SPLINE
SPL {X  -125.038, Y  +285.873, Z    +0.000, E1   +53.023, E3 +71876.787}
SPL {X  -149.949, Y  +329.886, Z    +0.000, E1   +41.515, E3 +71898.352}
SPL {X  -157.246, Y  +356.141, Z    +0.000, E1   +27.282, E3 +71903.408}
SPL {X  -159.525, Y  +373.376, Z    +0.000, E1   +13.812, E3 +71905.065}
SPL {X  -160.000, Y  +387.264, Z    +0.000, E1    +0.544, E3 +71905.523}
SPL {X  -160.000, Y  +390.384, Z    +0.000, E1    -6.008, E3 +71905.560}
SPL {X  -160.000, Y  +395.752, Z    +0.000, E1   -19.038, E3 +71905.754}
SPL {X  -160.000, Y  +404.289, Z    +0.000, E1   -38.292, E3 +71906.422}
SPL {X  -160.000, Y  +418.681, Z    +0.000, E1   -56.949, E3 +71908.612}
SPL {X  -160.000, Y  +471.977, Z    +0.000, E1   -70.792, E3 +71925.131}
SPL {X  -159.977, Y  +677.138, Z    +0.000, E1   -73.665, E3 +72021.623}
SPL {X  -157.805, Y  +700.810, Z    +0.000, E1   -73.511, E3 +72038.453}
SPL {X  -152.242, Y  +723.618, Z    +0.000, E1   -72.940, E3 +72058.366}
SPL {X  -145.929, Y  +740.010, Z    +0.000, E1   -72.229, E3 +72074.837}
SPL {X  -139.114, Y  +753.439, Z    +0.000, E1   -71.436, E3 +72089.476}
SPL {X  -132.333, Y  +764.333, Z    +0.000, E1   -70.535, E3 +72102.100}
SPL {X  -125.486, Y  +773.664, Z    +0.000, E1   -69.598, E3 +72113.074}
SPL {X  -121.321, Y  +778.713, Z    +0.000, E1   -68.872, E3 +72119.084}
SPL {X   -77.337, Y  +814.468, Z    +0.000, E1   -56.377, E3 +72237.715}
ENDSPLINE

SPLINE
SPL {X  -134.727, Y  +760.706, Z    +0.000, E1   -50.460, E3 +72425.947}
SPL {X  -155.580, Y  +711.748, Z    +0.000, E1   -32.084, E3 +72442.861}
SPL {X  -159.445, Y  +687.715, Z    +0.000, E1   -14.660, E3 +72445.708}
SPL {X  -159.995, Y  +675.725, Z    +0.000, E1    -3.424, E3 +72446.219}
SPL {X  -160.000, Y  +671.714, Z    +0.000, E1    +0.835, E3 +72446.259}
SPL {X  -160.000, Y  +663.084, Z    +0.000, E1   +21.134, E3 +72446.584}
SPL {X  -160.000, Y  +650.910, Z    +0.000, E1   +46.005, E3 +72447.738}
SPL {X  -160.000, Y  +634.843, Z    +0.000, E1   +61.273, E3 +72450.414}
SPL {X  -160.000, Y  +578.679, Z    +0.000, E1   +71.665, E3 +72468.248}
SPL {X  -160.000, Y  +387.528, Z    +0.000, E1   +73.487, E3 +72561.061}
SPL {X  -159.218, Y  +369.903, Z    +0.000, E1   +73.425, E3 +72572.928}
SPL {X  -156.808, Y  +353.900, Z    +0.000, E1   +73.180, E3 +72585.531}
SPL {X  -154.539, Y  +344.254, Z    +0.000, E1   +72.827, E3 +72595.069}
ENDSPLINE

SPLINE
SPL {X  -157.258, Y  +356.206, Z    +0.000, E1   +70.434, E3 +72609.641}
ENDSPLINE

SPLINE
SPL {X  -150.342, Y  +330.952, Z    +0.000, E1   +71.154, E3 +72621.314}
SPL {X  -141.358, Y  +310.748, Z    +0.000, E1   +71.233, E3 +72634.019}
SPL {X  -134.330, Y  +298.778, Z    +0.000, E1   +70.323, E3 +72647.867}
SPL {X  -128.957, Y  +290.989, Z    +0.000, E1   +69.528, E3 +72657.232}
SPL {X  -124.846, Y  +285.632, Z    +0.000, E1   +68.906, E3 +72663.695}
SPL {X  -121.783, Y  +281.927, Z    +0.000, E1   +68.403, E3 +72668.127}
SPL {X   -79.219, Y  +246.688, Z    +0.000, E1   +55.887, E3 +72789.634}
ENDSPLINE

SPLINE
SPL {X  -125.038, Y  +285.873, Z    +0.000, E1   +53.023, E3 +72966.675}
SPL {X  -149.949, Y  +329.886, Z    +0.000, E1   +41.515, E3 +72988.240}
SPL {X  -157.246, Y  +356.141, Z    +0.000, E1   +27.282, E3 +72993.296}
SPL {X  -159.525, Y  +373.376, Z    +0.000, E1   +13.812, E3 +72994.954}
SPL {X  -160.000, Y  +387.264, Z    +0.000, E1    +0.544, E3 +72995.411}
SPL {X  -160.000, Y  +390.384, Z    +0.000, E1    -6.008, E3 +72995.448}
SPL {X  -160.000, Y  +395.752, Z    +0.000, E1   -19.038, E3 +72995.642}
SPL {X  -160.000, Y  +404.289, Z    +0.000, E1   -38.292, E3 +72996.311}
SPL {X  -160.000, Y  +418.681, Z    +0.000, E1   -56.949, E3 +72998.500}
SPL {X  -160.000, Y  +471.977, Z    +0.000, E1   -70.792, E3 +73015.020}
SPL {X  -159.977, Y  +677.138, Z    +0.000, E1   -73.665, E3 +73111.511}
SPL {X  -157.805, Y  +700.810, Z    +0.000, E1   -73.511, E3 +73128.341}
SPL {X  -152.242, Y  +723.618, Z    +0.000, E1   -72.940, E3 +73148.254}
SPL {X  -145.929, Y  +740.010, Z    +0.000, E1   -72.229, E3 +73164.725}
SPL {X  -139.114, Y  +753.439, Z    +0.000, E1   -71.436, E3 +73179.364}
SPL {X  -132.333, Y  +764.333, Z    +0.000, E1   -70.535, E3 +73191.988}
SPL {X  -125.486, Y  +773.664, Z    +0.000, E1   -69.598, E3 +73202.962}
SPL {X  -121.321, Y  +778.713, Z    +0.000, E1   -68.872, E3 +73208.972}
SPL {X   -77.337, Y  +814.468, Z    +0.000, E1   -56.377, E3 +73327.603}
ENDSPLINE

SPLINE
SPL {X  -134.727, Y  +760.706, Z    +0.000, E1   -50.460, E3 +73515.835}
SPL {X  -155.580, Y  +711.748, Z    +0.000, E1   -32.084, E3 +73532.750}
SPL {X  -159.445, Y  +687.715, Z    +0.000, E1   -14.660, E3 +73535.596}
SPL {X  -159.995, Y  +675.725, Z    +0.000, E1    -3.424, E3 +73536.107}
SPL {X  -160.000, Y  +671.714, Z    +0.000, E1    +0.835, E3 +73536.148}
SPL {X  -160.000, Y  +663.084, Z    +0.000, E1   +21.134, E3 +73536.472}
SPL {X  -160.000, Y  +650.910, Z    +0.000, E1   +46.005, E3 +73537.626}
SPL {X  -160.000, Y  +634.843, Z    +0.000, E1   +61.273, E3 +73540.302}
SPL {X  -160.000, Y  +578.679, Z    +0.000, E1   +71.665, E3 +73558.136}
SPL {X  -160.000, Y  +387.528, Z    +0.000, E1   +73.487, E3 +73650.949}
SPL {X  -159.218, Y  +369.903, Z    +0.000, E1   +73.425, E3 +73662.816}
SPL {X  -156.808, Y  +353.900, Z    +0.000, E1   +73.180, E3 +73675.420}
SPL {X  -154.539, Y  +344.254, Z    +0.000, E1   +72.827, E3 +73684.957}
ENDSPLINE

SPLINE
SPL {X  -157.258, Y  +356.206, Z    +0.000, E1   +70.434, E3 +73699.529}
ENDSPLINE

SPLINE
SPL {X  -150.342, Y  +330.952, Z    +0.000, E1   +71.154, E3 +73711.202}
SPL {X  -141.358, Y  +310.748, Z    +0.000, E1   +71.233, E3 +73723.907}
SPL {X  -134.330, Y  +298.778, Z    +0.000, E1   +70.323, E3 +73737.755}
SPL {X  -128.957, Y  +290.989, Z    +0.000, E1   +69.528, E3 +73747.120}
SPL {X  -124.846, Y  +285.632, Z    +0.000, E1   +68.906, E3 +73753.583}
SPL {X  -121.783, Y  +281.927, Z    +0.000, E1   +68.403, E3 +73758.015}
SPL {X   -79.219, Y  +246.688, Z    +0.000, E1   +55.887, E3 +73879.522}
ENDSPLINE

SPLINE
SPL {X  -125.038, Y  +285.873, Z    +0.000, E1   +53.023, E3 +74056.563}
SPL {X  -149.949, Y  +329.886, Z    +0.000, E1   +41.515, E3 +74078.128}
SPL {X  -157.246, Y  +356.141, Z    +0.000, E1   +27.282, E3 +74083.184}
SPL {X  -159.525, Y  +373.376, Z    +0.000, E1   +13.812, E3 +74084.842}
SPL {X  -160.000, Y  +387.264, Z    +0.000, E1    +0.544, E3 +74085.299}
SPL {X  -160.000, Y  +390.384, Z    +0.000, E1    -6.008, E3 +74085.336}
SPL {X  -160.000, Y  +395.752, Z    +0.000, E1   -19.038, E3 +74085.530}
SPL {X  -160.000, Y  +404.289, Z    +0.000, E1   -38.292, E3 +74086.199}
SPL {X  -160.000, Y  +418.681, Z    +0.000, E1   -56.949, E3 +74088.388}
SPL {X  -160.000, Y  +471.977, Z    +0.000, E1   -70.792, E3 +74104.908}
SPL {X  -159.977, Y  +677.138, Z    +0.000, E1   -73.665, E3 +74201.399}
SPL {X  -157.805, Y  +700.810, Z    +0.000, E1   -73.511, E3 +74218.229}
SPL {X  -152.242, Y  +723.618, Z    +0.000, E1   -72.940, E3 +74238.142}
SPL {X  -145.929, Y  +740.010, Z    +0.000, E1   -72.229, E3 +74254.613}
SPL {X  -139.114, Y  +753.439, Z    +0.000, E1   -71.436, E3 +74269.252}
SPL {X  -132.333, Y  +764.333, Z    +0.000, E1   -70.535, E3 +74281.876}
SPL {X  -125.486, Y  +773.664, Z    +0.000, E1   -69.598, E3 +74292.850}
SPL {X  -121.321, Y  +778.713, Z    +0.000, E1   -68.872, E3 +74298.860}
SPL {X   -77.337, Y  +814.468, Z    +0.000, E1   -56.377, E3 +74417.491}
ENDSPLINE

SPLINE
SPL {X  -134.727, Y  +760.706, Z    +0.000, E1   -50.460, E3 +74605.723}
SPL {X  -155.580, Y  +711.748, Z    +0.000, E1   -32.084, E3 +74622.638}
SPL {X  -159.445, Y  +687.715, Z    +0.000, E1   -14.660, E3 +74625.484}
SPL {X  -159.995, Y  +675.725, Z    +0.000, E1    -3.424, E3 +74625.995}
SPL {X  -160.000, Y  +671.714, Z    +0.000, E1    +0.835, E3 +74626.036}
SPL {X  -160.000, Y  +663.084, Z    +0.000, E1   +21.134, E3 +74626.360}
SPL {X  -160.000, Y  +650.910, Z    +0.000, E1   +46.005, E3 +74627.514}
SPL {X  -160.000, Y  +634.843, Z    +0.000, E1   +61.273, E3 +74630.191}
SPL {X  -160.000, Y  +578.679, Z    +0.000, E1   +71.665, E3 +74648.024}
SPL {X  -160.000, Y  +387.528, Z    +0.000, E1   +73.487, E3 +74740.837}
SPL {X  -159.218, Y  +369.903, Z    +0.000, E1   +73.425, E3 +74752.704}
SPL {X  -156.808, Y  +353.900, Z    +0.000, E1   +73.180, E3 +74765.308}
SPL {X  -154.539, Y  +344.254, Z    +0.000, E1   +72.827, E3 +74774.845}
ENDSPLINE

SPLINE
SPL {X  -157.258, Y  +356.206, Z    +0.000, E1   +70.434, E3 +74789.417}
ENDSPLINE

SPLINE
SPL {X  -150.342, Y  +330.952, Z    +0.000, E1   +71.154, E3 +74801.090}
SPL {X  -141.358, Y  +310.748, Z    +0.000, E1   +71.233, E3 +74813.795}
SPL {X  -134.330, Y  +298.778, Z    +0.000, E1   +70.323, E3 +74827.643}
SPL {X  -128.957, Y  +290.989, Z    +0.000, E1   +69.528, E3 +74837.008}
SPL {X  -124.846, Y  +285.632, Z    +0.000, E1   +68.906, E3 +74843.471}
SPL {X  -121.783, Y  +281.927, Z    +0.000, E1   +68.403, E3 +74847.903}
SPL {X   -79.219, Y  +246.688, Z    +0.000, E1   +55.887, E3 +74969.410}
ENDSPLINE

SPLINE
SPL {X  -125.038, Y  +285.873, Z    +0.000, E1   +53.023, E3 +75146.451}
SPL {X  -149.949, Y  +329.886, Z    +0.000, E1   +41.515, E3 +75168.016}
SPL {X  -157.246, Y  +356.141, Z    +0.000, E1   +27.282, E3 +75173.073}
SPL {X  -159.525, Y  +373.376, Z    +0.000, E1   +13.812, E3 +75174.730}
SPL {X  -160.000, Y  +387.264, Z    +0.000, E1    +0.544, E3 +75175.187}
SPL {X  -160.000, Y  +390.384, Z    +0.000, E1    -6.008, E3 +75175.225}
SPL {X  -160.000, Y  +395.752, Z    +0.000, E1   -19.038, E3 +75175.418}
SPL {X  -160.000, Y  +404.289, Z    +0.000, E1   -38.292, E3 +75176.087}
SPL {X  -160.000, Y  +418.681, Z    +0.000, E1   -56.949, E3 +75178.276}
SPL {X  -160.000, Y  +471.977, Z    +0.000, E1   -70.792, E3 +75194.796}
SPL {X  -159.977, Y  +677.138, Z    +0.000, E1   -73.665, E3 +75291.287}
SPL {X  -157.805, Y  +700.810, Z    +0.000, E1   -73.511, E3 +75308.117}
SPL {X  -152.242, Y  +723.618, Z    +0.000, E1   -72.940, E3 +75328.030}
SPL {X  -145.929, Y  +740.010, Z    +0.000, E1   -72.229, E3 +75344.501}
SPL {X  -139.114, Y  +753.439, Z    +0.000, E1   -71.436, E3 +75359.140}
SPL {X  -132.333, Y  +764.333, Z    +0.000, E1   -70.535, E3 +75371.764}
SPL {X  -125.486, Y  +773.664, Z    +0.000, E1   -69.598, E3 +75382.738}
SPL {X  -121.321, Y  +778.713, Z    +0.000, E1   -68.872, E3 +75388.748}
SPL {X   -77.337, Y  +814.468, Z    +0.000, E1   -56.377, E3 +75507.379}
ENDSPLINE

SPLINE
SPL {X  -134.727, Y  +760.706, Z    +0.000, E1   -50.460, E3 +75695.611}
SPL {X  -155.580, Y  +711.748, Z    +0.000, E1   -32.084, E3 +75712.526}
SPL {X  -159.445, Y  +687.715, Z    +0.000, E1   -14.660, E3 +75715.372}
SPL {X  -159.995, Y  +675.725, Z    +0.000, E1    -3.424, E3 +75715.883}
SPL {X  -160.000, Y  +671.714, Z    +0.000, E1    +0.835, E3 +75715.924}
SPL {X  -160.000, Y  +663.084, Z    +0.000, E1   +21.134, E3 +75716.248}
SPL {X  -160.000, Y  +650.910, Z    +0.000, E1   +46.005, E3 +75717.402}
SPL {X  -160.000, Y  +634.843, Z    +0.000, E1   +61.273, E3 +75720.079}
SPL {X  -160.000, Y  +578.679, Z    +0.000, E1   +71.665, E3 +75737.912}
SPL {X  -160.000, Y  +387.528, Z    +0.000, E1   +73.487, E3 +75830.725}
SPL {X  -159.218, Y  +369.903, Z    +0.000, E1   +73.425, E3 +75842.592}
SPL {X  -156.808, Y  +353.900, Z    +0.000, E1   +73.180, E3 +75855.196}
SPL {X  -154.539, Y  +344.254, Z    +0.000, E1   +72.827, E3 +75864.733}
ENDSPLINE

SPLINE
SPL {X  -157.258, Y  +356.206, Z    +0.000, E1   +70.434, E3 +75879.305}
ENDSPLINE

SPLINE
SPL {X  -150.342, Y  +330.952, Z    +0.000, E1   +71.154, E3 +75890.978}
SPL {X  -141.358, Y  +310.748, Z    +0.000, E1   +71.233, E3 +75903.683}
SPL {X  -134.330, Y  +298.778, Z    +0.000, E1   +70.323, E3 +75917.531}
SPL {X  -128.957, Y  +290.989, Z    +0.000, E1   +69.528, E3 +75926.896}
SPL {X  -124.846, Y  +285.632, Z    +0.000, E1   +68.906, E3 +75933.359}
SPL {X  -121.783, Y  +281.927, Z    +0.000, E1   +68.403, E3 +75937.791}
SPL {X   -79.219, Y  +246.688, Z    +0.000, E1   +55.887, E3 +76059.298}
ENDSPLINE

SPLINE
SPL {X  -125.038, Y  +285.873, Z    +0.000, E1   +53.023, E3 +76236.339}
SPL {X  -149.949, Y  +329.886, Z    +0.000, E1   +41.515, E3 +76257.904}
SPL {X  -157.246, Y  +356.141, Z    +0.000, E1   +27.282, E3 +76262.961}
SPL {X  -159.525, Y  +373.376, Z    +0.000, E1   +13.812, E3 +76264.618}
SPL {X  -160.000, Y  +387.264, Z    +0.000, E1    +0.544, E3 +76265.075}
SPL {X  -160.000, Y  +390.384, Z    +0.000, E1    -6.008, E3 +76265.113}
SPL {X  -160.000, Y  +395.752, Z    +0.000, E1   -19.038, E3 +76265.306}
SPL {X  -160.000, Y  +404.289, Z    +0.000, E1   -38.292, E3 +76265.975}
SPL {X  -160.000, Y  +418.681, Z    +0.000, E1   -56.949, E3 +76268.164}
SPL {X  -160.000, Y  +458.961, Z    +0.000, E1   -69.778, E3 +76279.761}
SPL {X  -160.000, Y  +485.343, Z    +0.000, E1   -71.539, E3 +76289.747}
SPL {X  -159.977, Y  +677.138, Z    +0.000, E1   -73.665, E3 +76381.175}
SPL {X  -157.805, Y  +700.810, Z    +0.000, E1   -73.511, E3 +76398.005}
SPL {X  -152.242, Y  +723.618, Z    +0.000, E1   -72.940, E3 +76417.918}
SPL {X  -145.929, Y  +740.010, Z    +0.000, E1   -72.229, E3 +76434.389}
SPL {X  -139.114, Y  +753.439, Z    +0.000, E1   -71.436, E3 +76449.028}
SPL {X  -132.333, Y  +764.333, Z    +0.000, E1   -70.535, E3 +76461.652}
SPL {X  -125.486, Y  +773.664, Z    +0.000, E1   -69.598, E3 +76472.626}
SPL {X  -121.321, Y  +778.713, Z    +0.000, E1   -68.872, E3 +76478.636}
SPL {X   -77.337, Y  +814.468, Z    +0.000, E1   -56.377, E3 +76597.267}
ENDSPLINE

SPLINE
SPL {X  -134.727, Y  +760.706, Z    +0.000, E1   -50.460, E3 +76785.499}
SPL {X  -155.580, Y  +711.748, Z    +0.000, E1   -32.084, E3 +76802.414}
SPL {X  -159.445, Y  +687.715, Z    +0.000, E1   -14.660, E3 +76805.260}
SPL {X  -159.995, Y  +675.725, Z    +0.000, E1    -3.424, E3 +76805.771}
SPL {X  -160.000, Y  +671.714, Z    +0.000, E1    +0.835, E3 +76805.812}
SPL {X  -160.000, Y  +663.084, Z    +0.000, E1   +21.134, E3 +76806.136}
SPL {X  -160.000, Y  +650.910, Z    +0.000, E1   +46.005, E3 +76807.290}
SPL {X  -160.000, Y  +634.843, Z    +0.000, E1   +61.273, E3 +76809.967}
SPL {X  -160.000, Y  +578.679, Z    +0.000, E1   +71.665, E3 +76827.800}
SPL {X  -160.000, Y  +387.528, Z    +0.000, E1   +73.487, E3 +76920.613}
SPL {X  -159.218, Y  +369.903, Z    +0.000, E1   +73.425, E3 +76932.480}
SPL {X  -156.808, Y  +353.900, Z    +0.000, E1   +73.180, E3 +76945.084}
SPL {X  -154.539, Y  +344.254, Z    +0.000, E1   +72.827, E3 +76954.621}
ENDSPLINE

SPLINE
SPL {X  -157.258, Y  +356.206, Z    +0.000, E1   +70.434, E3 +76969.193}
ENDSPLINE

SPLINE
SPL {X  -150.342, Y  +330.952, Z    +0.000, E1   +71.154, E3 +76980.866}
SPL {X  -141.358, Y  +310.748, Z    +0.000, E1   +71.233, E3 +76993.572}
SPL {X  -134.330, Y  +298.778, Z    +0.000, E1   +70.323, E3 +77007.419}
SPL {X  -128.957, Y  +290.989, Z    +0.000, E1   +69.528, E3 +77016.784}
SPL {X  -124.846, Y  +285.632, Z    +0.000, E1   +68.906, E3 +77023.247}
SPL {X  -121.783, Y  +281.927, Z    +0.000, E1   +68.403, E3 +77027.679}
SPL {X   -79.219, Y  +246.688, Z    +0.000, E1   +55.887, E3 +77149.186}
ENDSPLINE

SPLINE
SPL {X  -125.038, Y  +285.873, Z    +0.000, E1   +53.023, E3 +77326.227}
SPL {X  -149.949, Y  +329.886, Z    +0.000, E1   +41.515, E3 +77347.792}
SPL {X  -157.246, Y  +356.141, Z    +0.000, E1   +27.282, E3 +77352.849}
SPL {X  -159.525, Y  +373.376, Z    +0.000, E1   +13.812, E3 +77354.506}
SPL {X  -160.000, Y  +387.264, Z    +0.000, E1    +0.544, E3 +77354.963}
SPL {X  -160.000, Y  +390.384, Z    +0.000, E1    -6.008, E3 +77355.001}
SPL {X  -160.000, Y  +395.752, Z    +0.000, E1   -19.038, E3 +77355.194}
SPL {X  -160.000, Y  +404.289, Z    +0.000, E1   -38.292, E3 +77355.863}
SPL {X  -160.000, Y  +418.681, Z    +0.000, E1   -56.949, E3 +77358.052}
SPL {X  -160.000, Y  +471.977, Z    +0.000, E1   -70.792, E3 +77374.572}
SPL {X  -159.977, Y  +677.138, Z    +0.000, E1   -73.665, E3 +77471.063}
SPL {X  -157.805, Y  +700.810, Z    +0.000, E1   -73.511, E3 +77487.893}
SPL {X  -152.242, Y  +723.618, Z    +0.000, E1   -72.940, E3 +77507.806}
SPL {X  -145.929, Y  +740.010, Z    +0.000, E1   -72.229, E3 +77524.277}
SPL {X  -139.114, Y  +753.439, Z    +0.000, E1   -71.436, E3 +77538.916}
SPL {X  -132.333, Y  +764.333, Z    +0.000, E1   -70.535, E3 +77551.540}
SPL {X  -125.486, Y  +773.664, Z    +0.000, E1   -69.598, E3 +77562.514}
SPL {X  -121.321, Y  +778.713, Z    +0.000, E1   -68.872, E3 +77568.524}
SPL {X   -77.337, Y  +814.468, Z    +0.000, E1   -56.377, E3 +77687.155}
ENDSPLINE

SPLINE
SPL {X  -134.727, Y  +760.706, Z    +0.000, E1   -50.460, E3 +77875.387}
SPL {X  -155.580, Y  +711.748, Z    +0.000, E1   -32.084, E3 +77892.302}
SPL {X  -159.445, Y  +687.715, Z    +0.000, E1   -14.660, E3 +77895.149}
SPL {X  -159.995, Y  +675.725, Z    +0.000, E1    -3.424, E3 +77895.659}
SPL {X  -160.000, Y  +671.714, Z    +0.000, E1    +0.835, E3 +77895.700}
SPL {X  -160.000, Y  +663.084, Z    +0.000, E1   +21.134, E3 +77896.024}
SPL {X  -160.000, Y  +650.910, Z    +0.000, E1   +46.005, E3 +77897.178}
SPL {X  -160.000, Y  +634.843, Z    +0.000, E1   +61.273, E3 +77899.855}
SPL {X  -160.000, Y  +578.679, Z    +0.000, E1   +71.665, E3 +77917.688}
SPL {X  -160.000, Y  +387.528, Z    +0.000, E1   +73.487, E3 +78010.501}
SPL {X  -159.218, Y  +369.903, Z    +0.000, E1   +73.425, E3 +78022.368}
SPL {X  -156.808, Y  +353.900, Z    +0.000, E1   +73.180, E3 +78034.972}
SPL {X  -154.539, Y  +344.254, Z    +0.000, E1   +72.827, E3 +78044.509}
ENDSPLINE

SPLINE
SPL {X  -157.258, Y  +356.206, Z    +0.000, E1   +70.434, E3 +78059.082}
ENDSPLINE

SPLINE
SPL {X  -150.342, Y  +330.952, Z    +0.000, E1   +71.154, E3 +78070.754}
SPL {X  -141.358, Y  +310.748, Z    +0.000, E1   +71.233, E3 +78083.460}
SPL {X  -134.330, Y  +298.778, Z    +0.000, E1   +70.323, E3 +78097.307}
SPL {X  -128.957, Y  +290.989, Z    +0.000, E1   +69.528, E3 +78106.672}
SPL {X  -124.846, Y  +285.632, Z    +0.000, E1   +68.906, E3 +78113.135}
SPL {X  -121.783, Y  +281.927, Z    +0.000, E1   +68.403, E3 +78117.568}
SPL {X   -79.219, Y  +246.688, Z    +0.000, E1   +55.887, E3 +78239.074}
ENDSPLINE

SPLINE
SPL {X  -125.038, Y  +285.873, Z    +0.000, E1   +53.023, E3 +78416.115}
SPL {X  -149.949, Y  +329.886, Z    +0.000, E1   +41.515, E3 +78437.680}
SPL {X  -157.246, Y  +356.141, Z    +0.000, E1   +27.282, E3 +78442.737}
SPL {X  -159.525, Y  +373.376, Z    +0.000, E1   +13.812, E3 +78444.394}
SPL {X  -160.000, Y  +387.264, Z    +0.000, E1    +0.544, E3 +78444.851}
SPL {X  -160.000, Y  +390.384, Z    +0.000, E1    -6.008, E3 +78444.889}
SPL {X  -160.000, Y  +395.752, Z    +0.000, E1   -19.038, E3 +78445.082}
SPL {X  -160.000, Y  +404.289, Z    +0.000, E1   -38.292, E3 +78445.751}
SPL {X  -160.000, Y  +418.681, Z    +0.000, E1   -56.949, E3 +78447.940}
SPL {X  -160.000, Y  +471.977, Z    +0.000, E1   -70.792, E3 +78464.460}
SPL {X  -159.977, Y  +677.138, Z    +0.000, E1   -73.665, E3 +78560.951}
SPL {X  -157.805, Y  +700.810, Z    +0.000, E1   -73.511, E3 +78577.781}
SPL {X  -152.242, Y  +723.618, Z    +0.000, E1   -72.940, E3 +78597.694}
SPL {X  -145.929, Y  +740.010, Z    +0.000, E1   -72.229, E3 +78614.165}
SPL {X  -139.114, Y  +753.439, Z    +0.000, E1   -71.436, E3 +78628.804}
SPL {X  -132.333, Y  +764.333, Z    +0.000, E1   -70.535, E3 +78641.428}
SPL {X  -125.486, Y  +773.664, Z    +0.000, E1   -69.598, E3 +78652.402}
SPL {X  -121.321, Y  +778.713, Z    +0.000, E1   -68.872, E3 +78658.412}
SPL {X   -77.337, Y  +814.468, Z    +0.000, E1   -56.377, E3 +78777.043}
ENDSPLINE

SPLINE
SPL {X  -134.727, Y  +760.706, Z    +0.000, E1   -50.460, E3 +78965.275}
SPL {X  -155.580, Y  +711.748, Z    +0.000, E1   -32.084, E3 +78982.190}
SPL {X  -159.445, Y  +687.715, Z    +0.000, E1   -14.660, E3 +78985.037}
SPL {X  -159.995, Y  +675.725, Z    +0.000, E1    -3.424, E3 +78985.547}
SPL {X  -160.000, Y  +671.714, Z    +0.000, E1    +0.835, E3 +78985.588}
SPL {X  -160.000, Y  +663.084, Z    +0.000, E1   +21.134, E3 +78985.912}
SPL {X  -160.000, Y  +650.910, Z    +0.000, E1   +46.005, E3 +78987.066}
SPL {X  -160.000, Y  +634.843, Z    +0.000, E1   +61.273, E3 +78989.743}
SPL {X  -160.000, Y  +578.679, Z    +0.000, E1   +71.665, E3 +79007.576}
SPL {X  -160.000, Y  +387.528, Z    +0.000, E1   +73.487, E3 +79100.389}
SPL {X  -159.218, Y  +369.903, Z    +0.000, E1   +73.425, E3 +79112.256}
SPL {X  -156.808, Y  +353.900, Z    +0.000, E1   +73.180, E3 +79124.860}
SPL {X  -154.539, Y  +344.254, Z    +0.000, E1   +72.827, E3 +79134.397}
ENDSPLINE

SPLINE
SPL {X  -157.258, Y  +356.206, Z    +0.000, E1   +70.434, E3 +79148.970}
ENDSPLINE

SPLINE
SPL {X  -150.342, Y  +330.952, Z    +0.000, E1   +71.154, E3 +79160.642}
SPL {X  -141.358, Y  +310.748, Z    +0.000, E1   +71.233, E3 +79173.348}
SPL {X  -134.330, Y  +298.778, Z    +0.000, E1   +70.323, E3 +79187.195}
SPL {X  -128.957, Y  +290.989, Z    +0.000, E1   +69.528, E3 +79196.560}
SPL {X  -124.846, Y  +285.632, Z    +0.000, E1   +68.906, E3 +79203.023}
SPL {X  -121.783, Y  +281.927, Z    +0.000, E1   +68.403, E3 +79207.456}
SPL {X   -79.219, Y  +246.688, Z    +0.000, E1   +55.887, E3 +79328.962}
ENDSPLINE

SPLINE
SPL {X  -125.038, Y  +285.873, Z    +0.000, E1   +53.023, E3 +79506.003}
SPL {X  -149.949, Y  +329.886, Z    +0.000, E1   +41.515, E3 +79527.568}
SPL {X  -157.246, Y  +356.141, Z    +0.000, E1   +27.282, E3 +79532.625}
SPL {X  -159.525, Y  +373.376, Z    +0.000, E1   +13.812, E3 +79534.282}
SPL {X  -160.000, Y  +387.264, Z    +0.000, E1    +0.544, E3 +79534.740}
SPL {X  -160.000, Y  +390.384, Z    +0.000, E1    -6.008, E3 +79534.777}
SPL {X  -160.000, Y  +395.752, Z    +0.000, E1   -19.038, E3 +79534.970}
SPL {X  -160.000, Y  +404.289, Z    +0.000, E1   -38.292, E3 +79535.639}
SPL {X  -160.000, Y  +418.681, Z    +0.000, E1   -56.949, E3 +79537.828}
SPL {X  -160.000, Y  +471.977, Z    +0.000, E1   -70.792, E3 +79554.348}
SPL {X  -159.977, Y  +677.138, Z    +0.000, E1   -73.665, E3 +79650.839}
SPL {X  -157.805, Y  +700.810, Z    +0.000, E1   -73.511, E3 +79667.669}
SPL {X  -152.242, Y  +723.618, Z    +0.000, E1   -72.940, E3 +79687.582}
SPL {X  -145.929, Y  +740.010, Z    +0.000, E1   -72.229, E3 +79704.053}
SPL {X  -139.114, Y  +753.439, Z    +0.000, E1   -71.436, E3 +79718.692}
SPL {X  -132.333, Y  +764.333, Z    +0.000, E1   -70.535, E3 +79731.316}
SPL {X  -125.486, Y  +773.664, Z    +0.000, E1   -69.598, E3 +79742.290}
SPL {X  -121.321, Y  +778.713, Z    +0.000, E1   -68.872, E3 +79748.300}
SPL {X   -77.337, Y  +814.468, Z    +0.000, E1   -56.377, E3 +79866.931}
ENDSPLINE

SPLINE
SPL {X  -134.727, Y  +760.706, Z    +0.000, E1   -50.460, E3 +80055.163}
SPL {X  -155.580, Y  +711.748, Z    +0.000, E1   -32.084, E3 +80072.078}
SPL {X  -159.445, Y  +687.715, Z    +0.000, E1   -14.660, E3 +80074.925}
SPL {X  -159.995, Y  +675.725, Z    +0.000, E1    -3.424, E3 +80075.435}
SPL {X  -160.000, Y  +671.714, Z    +0.000, E1    +0.835, E3 +80075.476}
SPL {X  -160.000, Y  +663.084, Z    +0.000, E1   +21.134, E3 +80075.800}
SPL {X  -160.000, Y  +650.910, Z    +0.000, E1   +46.005, E3 +80076.954}
SPL {X  -160.000, Y  +634.843, Z    +0.000, E1   +61.273, E3 +80079.631}
SPL {X  -160.000, Y  +578.679, Z    +0.000, E1   +71.665, E3 +80097.464}
SPL {X  -160.000, Y  +387.528, Z    +0.000, E1   +73.487, E3 +80190.277}
SPL {X  -159.218, Y  +369.903, Z    +0.000, E1   +73.425, E3 +80202.144}
SPL {X  -156.808, Y  +353.900, Z    +0.000, E1   +73.180, E3 +80214.748}
SPL {X  -154.539, Y  +344.254, Z    +0.000, E1   +72.827, E3 +80224.285}
ENDSPLINE

SPLINE
SPL {X  -157.258, Y  +356.206, Z    +0.000, E1   +70.434, E3 +80238.858}
ENDSPLINE

SPLINE
SPL {X  -150.342, Y  +330.952, Z    +0.000, E1   +71.154, E3 +80250.530}
SPL {X  -141.358, Y  +310.748, Z    +0.000, E1   +71.233, E3 +80263.236}
SPL {X  -134.330, Y  +298.778, Z    +0.000, E1   +70.323, E3 +80277.083}
SPL {X  -128.957, Y  +290.989, Z    +0.000, E1   +69.528, E3 +80286.448}
SPL {X  -124.846, Y  +285.632, Z    +0.000, E1   +68.906, E3 +80292.911}
SPL {X  -121.783, Y  +281.927, Z    +0.000, E1   +68.403, E3 +80297.344}
SPL {X   -79.219, Y  +246.688, Z    +0.000, E1   +55.887, E3 +80418.850}
ENDSPLINE

SPLINE
SPL {X  -125.038, Y  +285.873, Z    +0.000, E1   +53.023, E3 +80595.891}
SPL {X  -149.949, Y  +329.886, Z    +0.000, E1   +41.515, E3 +80617.456}
SPL {X  -157.246, Y  +356.141, Z    +0.000, E1   +27.282, E3 +80622.513}
SPL {X  -159.525, Y  +373.376, Z    +0.000, E1   +13.812, E3 +80624.170}
SPL {X  -160.000, Y  +387.264, Z    +0.000, E1    +0.544, E3 +80624.628}
SPL {X  -160.000, Y  +390.384, Z    +0.000, E1    -6.008, E3 +80624.665}
SPL {X  -160.000, Y  +395.752, Z    +0.000, E1   -19.038, E3 +80624.858}
SPL {X  -160.000, Y  +404.289, Z    +0.000, E1   -38.292, E3 +80625.527}
SPL {X  -160.000, Y  +418.681, Z    +0.000, E1   -56.949, E3 +80627.717}
SPL {X  -160.000, Y  +471.977, Z    +0.000, E1   -70.792, E3 +80644.236}
SPL {X  -159.977, Y  +677.138, Z    +0.000, E1   -73.665, E3 +80740.727}
SPL {X  -157.805, Y  +700.810, Z    +0.000, E1   -73.511, E3 +80757.557}
SPL {X  -152.242, Y  +723.618, Z    +0.000, E1   -72.940, E3 +80777.470}
SPL {X  -145.929, Y  +740.010, Z    +0.000, E1   -72.229, E3 +80793.941}
SPL {X  -139.114, Y  +753.439, Z    +0.000, E1   -71.436, E3 +80808.580}
SPL {X  -132.333, Y  +764.333, Z    +0.000, E1   -70.535, E3 +80821.204}
SPL {X  -125.486, Y  +773.664, Z    +0.000, E1   -69.598, E3 +80832.178}
SPL {X  -121.321, Y  +778.713, Z    +0.000, E1   -68.872, E3 +80838.188}
SPL {X   -77.337, Y  +814.468, Z    +0.000, E1   -56.377, E3 +80956.819}
ENDSPLINE

SPLINE
SPL {X  -134.727, Y  +760.706, Z    +0.000, E1   -50.460, E3 +81145.051}
SPL {X  -155.580, Y  +711.748, Z    +0.000, E1   -32.084, E3 +81161.966}
SPL {X  -159.445, Y  +687.715, Z    +0.000, E1   -14.660, E3 +81164.813}
SPL {X  -159.995, Y  +675.725, Z    +0.000, E1    -3.424, E3 +81165.323}
SPL {X  -160.000, Y  +671.714, Z    +0.000, E1    +0.835, E3 +81165.364}
SPL {X  -160.000, Y  +663.084, Z    +0.000, E1   +21.134, E3 +81165.688}
SPL {X  -160.000, Y  +650.910, Z    +0.000, E1   +46.005, E3 +81166.842}
SPL {X  -160.000, Y  +634.843, Z    +0.000, E1   +61.273, E3 +81169.519}
SPL {X  -160.000, Y  +578.679, Z    +0.000, E1   +71.665, E3 +81187.352}
SPL {X  -160.000, Y  +387.528, Z    +0.000, E1   +73.487, E3 +81280.165}
SPL {X  -159.218, Y  +369.903, Z    +0.000, E1   +73.425, E3 +81292.032}
SPL {X  -156.808, Y  +353.900, Z    +0.000, E1   +73.180, E3 +81304.636}
SPL {X  -154.539, Y  +344.254, Z    +0.000, E1   +72.827, E3 +81314.173}
ENDSPLINE

SPLINE
SPL {X  -157.258, Y  +356.206, Z    +0.000, E1   +70.434, E3 +81328.746}
ENDSPLINE

SPLINE
SPL {X  -150.342, Y  +330.952, Z    +0.000, E1   +71.154, E3 +81340.418}
SPL {X  -141.358, Y  +310.748, Z    +0.000, E1   +71.233, E3 +81353.124}
SPL {X  -134.330, Y  +298.778, Z    +0.000, E1   +70.323, E3 +81366.971}
SPL {X  -128.957, Y  +290.989, Z    +0.000, E1   +69.528, E3 +81376.336}
SPL {X  -124.846, Y  +285.632, Z    +0.000, E1   +68.906, E3 +81382.799}
SPL {X  -121.783, Y  +281.927, Z    +0.000, E1   +68.403, E3 +81387.232}
SPL {X   -79.219, Y  +246.688, Z    +0.000, E1   +55.887, E3 +81508.738}
ENDSPLINE

SPLINE
SPL {X  -125.038, Y  +285.873, Z    +0.000, E1   +53.023, E3 +81685.779}
SPL {X  -149.949, Y  +329.886, Z    +0.000, E1   +41.515, E3 +81707.344}
SPL {X  -157.246, Y  +356.141, Z    +0.000, E1   +27.282, E3 +81712.401}
SPL {X  -159.525, Y  +373.376, Z    +0.000, E1   +13.812, E3 +81714.058}
SPL {X  -160.000, Y  +387.264, Z    +0.000, E1    +0.544, E3 +81714.516}
SPL {X  -160.000, Y  +390.384, Z    +0.000, E1    -6.008, E3 +81714.553}
SPL {X  -160.000, Y  +395.752, Z    +0.000, E1   -19.038, E3 +81714.746}
SPL {X  -160.000, Y  +404.289, Z    +0.000, E1   -38.292, E3 +81715.415}
SPL {X  -160.000, Y  +418.681, Z    +0.000, E1   -56.949, E3 +81717.605}
SPL {X  -160.000, Y  +471.977, Z    +0.000, E1   -70.792, E3 +81734.124}
SPL {X  -159.977, Y  +677.138, Z    +0.000, E1   -73.665, E3 +81830.615}
SPL {X  -157.805, Y  +700.810, Z    +0.000, E1   -73.511, E3 +81847.445}
SPL {X  -152.242, Y  +723.618, Z    +0.000, E1   -72.940, E3 +81867.358}
SPL {X  -145.929, Y  +740.010, Z    +0.000, E1   -72.229, E3 +81883.829}
SPL {X  -139.114, Y  +753.439, Z    +0.000, E1   -71.436, E3 +81898.468}
SPL {X  -132.333, Y  +764.333, Z    +0.000, E1   -70.535, E3 +81911.092}
SPL {X  -125.486, Y  +773.664, Z    +0.000, E1   -69.598, E3 +81922.066}
SPL {X  -121.321, Y  +778.713, Z    +0.000, E1   -68.872, E3 +81928.076}
SPL {X   -77.337, Y  +814.468, Z    +0.000, E1   -56.377, E3 +82046.707}
ENDSPLINE

SPLINE
SPL {X  -134.727, Y  +760.706, Z    +0.000, E1   -50.460, E3 +82234.939}
SPL {X  -155.580, Y  +711.748, Z    +0.000, E1   -32.084, E3 +82251.854}
SPL {X  -159.445, Y  +687.715, Z    +0.000, E1   -14.660, E3 +82254.701}
SPL {X  -159.995, Y  +675.725, Z    +0.000, E1    -3.424, E3 +82255.211}
SPL {X  -160.000, Y  +671.714, Z    +0.000, E1    +0.835, E3 +82255.252}
SPL {X  -160.000, Y  +663.084, Z    +0.000, E1   +21.134, E3 +82255.576}
SPL {X  -160.000, Y  +650.910, Z    +0.000, E1   +46.005, E3 +82256.730}
SPL {X  -160.000, Y  +634.843, Z    +0.000, E1   +61.273, E3 +82259.407}
SPL {X  -160.000, Y  +578.679, Z    +0.000, E1   +71.665, E3 +82277.241}
SPL {X  -160.000, Y  +387.528, Z    +0.000, E1   +73.487, E3 +82370.053}
SPL {X  -159.218, Y  +369.903, Z    +0.000, E1   +73.425, E3 +82381.920}
SPL {X  -156.808, Y  +353.900, Z    +0.000, E1   +73.180, E3 +82394.524}
SPL {X  -154.539, Y  +344.254, Z    +0.000, E1   +72.827, E3 +82404.061}
ENDSPLINE

SPLINE
SPL {X  -157.258, Y  +356.206, Z    +0.000, E1   +70.434, E3 +82418.634}
ENDSPLINE

SPLINE
SPL {X  -150.342, Y  +330.952, Z    +0.000, E1   +71.154, E3 +82430.306}
SPL {X  -141.358, Y  +310.748, Z    +0.000, E1   +71.233, E3 +82443.012}
SPL {X  -134.330, Y  +298.778, Z    +0.000, E1   +70.323, E3 +82456.859}
SPL {X  -128.957, Y  +290.989, Z    +0.000, E1   +69.528, E3 +82466.224}
SPL {X  -124.846, Y  +285.632, Z    +0.000, E1   +68.906, E3 +82472.687}
SPL {X  -121.783, Y  +281.927, Z    +0.000, E1   +68.403, E3 +82477.120}
SPL {X   -79.219, Y  +246.688, Z    +0.000, E1   +55.887, E3 +82598.626}
ENDSPLINE

SPLINE
SPL {X  -125.038, Y  +285.873, Z    +0.000, E1   +53.023, E3 +82775.667}
SPL {X  -149.949, Y  +329.886, Z    +0.000, E1   +41.515, E3 +82797.232}
SPL {X  -157.246, Y  +356.141, Z    +0.000, E1   +27.282, E3 +82802.289}
SPL {X  -159.525, Y  +373.376, Z    +0.000, E1   +13.812, E3 +82803.946}
SPL {X  -160.000, Y  +387.264, Z    +0.000, E1    +0.544, E3 +82804.404}
SPL {X  -160.000, Y  +390.384, Z    +0.000, E1    -6.008, E3 +82804.441}
SPL {X  -160.000, Y  +395.752, Z    +0.000, E1   -19.038, E3 +82804.634}
SPL {X  -160.000, Y  +404.289, Z    +0.000, E1   -38.292, E3 +82805.303}
SPL {X  -160.000, Y  +418.681, Z    +0.000, E1   -56.949, E3 +82807.493}
SPL {X  -160.000, Y  +471.977, Z    +0.000, E1   -70.792, E3 +82824.012}
SPL {X  -159.977, Y  +677.138, Z    +0.000, E1   -73.665, E3 +82920.503}
SPL {X  -157.805, Y  +700.810, Z    +0.000, E1   -73.511, E3 +82937.333}
SPL {X  -152.242, Y  +723.618, Z    +0.000, E1   -72.940, E3 +82957.246}
SPL {X  -145.929, Y  +740.010, Z    +0.000, E1   -72.229, E3 +82973.717}
SPL {X  -139.114, Y  +753.439, Z    +0.000, E1   -71.436, E3 +82988.356}
SPL {X  -132.333, Y  +764.333, Z    +0.000, E1   -70.535, E3 +83000.980}
SPL {X  -125.486, Y  +773.664, Z    +0.000, E1   -69.598, E3 +83011.954}
SPL {X  -121.321, Y  +778.713, Z    +0.000, E1   -68.872, E3 +83017.964}
SPL {X   -77.337, Y  +814.468, Z    +0.000, E1   -56.377, E3 +83136.595}
ENDSPLINE

SPLINE
SPL {X  -134.727, Y  +760.706, Z    +0.000, E1   -50.460, E3 +83324.827}
SPL {X  -155.580, Y  +711.748, Z    +0.000, E1   -32.084, E3 +83341.742}
SPL {X  -159.445, Y  +687.715, Z    +0.000, E1   -14.660, E3 +83344.589}
SPL {X  -159.995, Y  +675.725, Z    +0.000, E1    -3.424, E3 +83345.099}
SPL {X  -160.000, Y  +671.714, Z    +0.000, E1    +0.835, E3 +83345.140}
SPL {X  -160.000, Y  +663.084, Z    +0.000, E1   +21.134, E3 +83345.464}
SPL {X  -160.000, Y  +650.910, Z    +0.000, E1   +46.005, E3 +83346.618}
SPL {X  -160.000, Y  +634.843, Z    +0.000, E1   +61.273, E3 +83349.295}
SPL {X  -160.000, Y  +578.679, Z    +0.000, E1   +71.665, E3 +83367.129}
SPL {X  -160.000, Y  +387.528, Z    +0.000, E1   +73.487, E3 +83459.941}
SPL {X  -159.218, Y  +369.903, Z    +0.000, E1   +73.425, E3 +83471.808}
SPL {X  -156.808, Y  +353.900, Z    +0.000, E1   +73.180, E3 +83484.412}
SPL {X  -154.539, Y  +344.254, Z    +0.000, E1   +72.827, E3 +83493.949}
ENDSPLINE

SPLINE
SPL {X  -157.258, Y  +356.206, Z    +0.000, E1   +70.434, E3 +83508.522}
ENDSPLINE

SPLINE
SPL {X  -150.342, Y  +330.952, Z    +0.000, E1   +71.154, E3 +83520.194}
SPL {X  -141.358, Y  +310.748, Z    +0.000, E1   +71.233, E3 +83532.900}
SPL {X  -134.330, Y  +298.778, Z    +0.000, E1   +70.323, E3 +83546.747}
SPL {X  -128.957, Y  +290.989, Z    +0.000, E1   +69.528, E3 +83556.112}
SPL {X  -124.846, Y  +285.632, Z    +0.000, E1   +68.906, E3 +83562.575}
SPL {X  -121.783, Y  +281.927, Z    +0.000, E1   +68.403, E3 +83567.008}
SPL {X   -79.219, Y  +246.688, Z    +0.000, E1   +55.887, E3 +83688.514}
ENDSPLINE

SPLINE
SPL {X  -125.038, Y  +285.873, Z    +0.000, E1   +53.023, E3 +83865.555}
SPL {X  -149.949, Y  +329.886, Z    +0.000, E1   +41.515, E3 +83887.120}
SPL {X  -157.246, Y  +356.141, Z    +0.000, E1   +27.282, E3 +83892.177}
SPL {X  -159.525, Y  +373.376, Z    +0.000, E1   +13.812, E3 +83893.834}
SPL {X  -160.000, Y  +387.264, Z    +0.000, E1    +0.544, E3 +83894.292}
SPL {X  -160.000, Y  +390.384, Z    +0.000, E1    -6.008, E3 +83894.329}
SPL {X  -160.000, Y  +395.752, Z    +0.000, E1   -19.038, E3 +83894.522}
SPL {X  -160.000, Y  +404.289, Z    +0.000, E1   -38.292, E3 +83895.191}
SPL {X  -160.000, Y  +418.681, Z    +0.000, E1   -56.949, E3 +83897.381}
SPL {X  -160.000, Y  +471.977, Z    +0.000, E1   -70.792, E3 +83913.900}
SPL {X  -159.977, Y  +677.138, Z    +0.000, E1   -73.665, E3 +84010.391}
SPL {X  -157.805, Y  +700.810, Z    +0.000, E1   -73.511, E3 +84027.221}
SPL {X  -152.242, Y  +723.618, Z    +0.000, E1   -72.940, E3 +84047.134}
SPL {X  -145.929, Y  +740.010, Z    +0.000, E1   -72.229, E3 +84063.605}
SPL {X  -139.114, Y  +753.439, Z    +0.000, E1   -71.436, E3 +84078.244}
SPL {X  -132.333, Y  +764.333, Z    +0.000, E1   -70.535, E3 +84090.868}
SPL {X  -125.486, Y  +773.664, Z    +0.000, E1   -69.598, E3 +84101.842}
SPL {X  -121.321, Y  +778.713, Z    +0.000, E1   -68.872, E3 +84107.852}
SPL {X   -77.337, Y  +814.468, Z    +0.000, E1   -56.377, E3 +84226.483}
ENDSPLINE

SPLINE
SPL {X  -134.727, Y  +760.706, Z    +0.000, E1   -50.460, E3 +84414.715}
SPL {X  -155.580, Y  +711.748, Z    +0.000, E1   -32.084, E3 +84431.630}
SPL {X  -159.445, Y  +687.715, Z    +0.000, E1   -14.660, E3 +84434.477}
SPL {X  -159.995, Y  +675.725, Z    +0.000, E1    -3.424, E3 +84434.988}
SPL {X  -160.000, Y  +671.714, Z    +0.000, E1    +0.835, E3 +84435.028}
SPL {X  -160.000, Y  +663.084, Z    +0.000, E1   +21.134, E3 +84435.352}
SPL {X  -160.000, Y  +650.910, Z    +0.000, E1   +46.005, E3 +84436.506}
SPL {X  -160.000, Y  +634.843, Z    +0.000, E1   +61.273, E3 +84439.183}
SPL {X  -160.000, Y  +578.679, Z    +0.000, E1   +71.665, E3 +84457.017}
SPL {X  -160.000, Y  +387.528, Z    +0.000, E1   +73.487, E3 +84549.829}
SPL {X  -159.218, Y  +369.903, Z    +0.000, E1   +73.425, E3 +84561.696}
SPL {X  -156.808, Y  +353.900, Z    +0.000, E1   +73.180, E3 +84574.300}
SPL {X  -154.539, Y  +344.254, Z    +0.000, E1   +72.827, E3 +84583.837}
ENDSPLINE

SPLINE
SPL {X  -157.258, Y  +356.206, Z    +0.000, E1   +70.434, E3 +84598.410}
ENDSPLINE

SPLINE
SPL {X  -150.342, Y  +330.952, Z    +0.000, E1   +71.154, E3 +84610.082}
SPL {X  -141.358, Y  +310.748, Z    +0.000, E1   +71.233, E3 +84622.788}
SPL {X  -134.330, Y  +298.778, Z    +0.000, E1   +70.323, E3 +84636.635}
SPL {X  -128.957, Y  +290.989, Z    +0.000, E1   +69.528, E3 +84646.000}
SPL {X  -124.846, Y  +285.632, Z    +0.000, E1   +68.906, E3 +84652.464}
SPL {X  -121.783, Y  +281.927, Z    +0.000, E1   +68.403, E3 +84656.896}
SPL {X   -79.219, Y  +246.688, Z    +0.000, E1   +55.887, E3 +84778.402}
ENDSPLINE

SPLINE
SPL {X  -125.038, Y  +285.873, Z    +0.000, E1   +53.023, E3 +84955.443}
SPL {X  -149.949, Y  +329.886, Z    +0.000, E1   +41.515, E3 +84977.008}
SPL {X  -157.246, Y  +356.141, Z    +0.000, E1   +27.282, E3 +84982.065}
SPL {X  -159.525, Y  +373.376, Z    +0.000, E1   +13.812, E3 +84983.722}
SPL {X  -160.000, Y  +387.264, Z    +0.000, E1    +0.544, E3 +84984.180}
SPL {X  -160.000, Y  +390.384, Z    +0.000, E1    -6.008, E3 +84984.217}
SPL {X  -160.000, Y  +395.752, Z    +0.000, E1   -19.038, E3 +84984.411}
SPL {X  -160.000, Y  +404.289, Z    +0.000, E1   -38.292, E3 +84985.079}
SPL {X  -160.000, Y  +418.681, Z    +0.000, E1   -56.949, E3 +84987.269}
SPL {X  -160.000, Y  +471.977, Z    +0.000, E1   -70.792, E3 +85003.788}
SPL {X  -159.977, Y  +677.138, Z    +0.000, E1   -73.665, E3 +85100.279}
SPL {X  -157.805, Y  +700.810, Z    +0.000, E1   -73.511, E3 +85117.109}
SPL {X  -152.242, Y  +723.618, Z    +0.000, E1   -72.940, E3 +85137.022}
SPL {X  -145.929, Y  +740.010, Z    +0.000, E1   -72.229, E3 +85153.494}
SPL {X  -139.114, Y  +753.439, Z    +0.000, E1   -71.436, E3 +85168.132}
SPL {X  -132.333, Y  +764.333, Z    +0.000, E1   -70.535, E3 +85180.756}
SPL {X  -125.486, Y  +773.664, Z    +0.000, E1   -69.598, E3 +85191.730}
SPL {X  -121.321, Y  +778.713, Z    +0.000, E1   -68.872, E3 +85197.740}
SPL {X   -77.337, Y  +814.468, Z    +0.000, E1   -56.377, E3 +85316.371}
ENDSPLINE

SPLINE
SPL {X  -134.727, Y  +760.706, Z    +0.000, E1   -50.460, E3 +85504.603}
SPL {X  -155.580, Y  +711.748, Z    +0.000, E1   -32.084, E3 +85521.518}
SPL {X  -159.445, Y  +687.715, Z    +0.000, E1   -14.660, E3 +85524.365}
SPL {X  -159.995, Y  +675.725, Z    +0.000, E1    -3.424, E3 +85524.876}
SPL {X  -160.000, Y  +671.714, Z    +0.000, E1    +0.835, E3 +85524.916}
SPL {X  -160.000, Y  +663.084, Z    +0.000, E1   +21.134, E3 +85525.240}
SPL {X  -160.000, Y  +650.910, Z    +0.000, E1   +46.005, E3 +85526.394}
SPL {X  -160.000, Y  +634.843, Z    +0.000, E1   +61.273, E3 +85529.071}
SPL {X  -160.000, Y  +578.679, Z    +0.000, E1   +71.665, E3 +85546.905}
SPL {X  -160.000, Y  +387.528, Z    +0.000, E1   +73.487, E3 +85639.717}
SPL {X  -159.218, Y  +369.903, Z    +0.000, E1   +73.425, E3 +85651.584}
SPL {X  -156.808, Y  +353.900, Z    +0.000, E1   +73.180, E3 +85664.188}
SPL {X  -154.539, Y  +344.254, Z    +0.000, E1   +72.827, E3 +85673.725}
ENDSPLINE

SPLINE
SPL {X  -157.258, Y  +356.206, Z    +0.000, E1   +70.434, E3 +85688.298}
ENDSPLINE

SPLINE
SPL {X  -150.342, Y  +330.952, Z    +0.000, E1   +71.154, E3 +85699.970}
SPL {X  -141.358, Y  +310.748, Z    +0.000, E1   +71.233, E3 +85712.676}
SPL {X  -134.330, Y  +298.778, Z    +0.000, E1   +70.323, E3 +85726.523}
SPL {X  -128.957, Y  +290.989, Z    +0.000, E1   +69.528, E3 +85735.888}
SPL {X  -124.846, Y  +285.632, Z    +0.000, E1   +68.906, E3 +85742.352}
SPL {X  -121.783, Y  +281.927, Z    +0.000, E1   +68.403, E3 +85746.784}
SPL {X   -79.219, Y  +246.688, Z    +0.000, E1   +55.887, E3 +85868.290}
ENDSPLINE

SPLINE
SPL {X  -125.038, Y  +285.873, Z    +0.000, E1   +53.023, E3 +86045.331}
SPL {X  -149.949, Y  +329.886, Z    +0.000, E1   +41.515, E3 +86066.896}
SPL {X  -157.246, Y  +356.141, Z    +0.000, E1   +27.282, E3 +86071.953}
SPL {X  -159.525, Y  +373.376, Z    +0.000, E1   +13.812, E3 +86073.610}
SPL {X  -160.000, Y  +387.264, Z    +0.000, E1    +0.544, E3 +86074.068}
SPL {X  -160.000, Y  +390.384, Z    +0.000, E1    -6.008, E3 +86074.105}
SPL {X  -160.000, Y  +395.752, Z    +0.000, E1   -19.038, E3 +86074.299}
SPL {X  -160.000, Y  +404.289, Z    +0.000, E1   -38.292, E3 +86074.967}
SPL {X  -160.000, Y  +418.681, Z    +0.000, E1   -56.949, E3 +86077.157}
SPL {X  -160.000, Y  +471.977, Z    +0.000, E1   -70.792, E3 +86093.676}
SPL {X  -159.977, Y  +677.138, Z    +0.000, E1   -73.665, E3 +86190.167}
SPL {X  -157.805, Y  +700.810, Z    +0.000, E1   -73.511, E3 +86206.997}
SPL {X  -152.242, Y  +723.618, Z    +0.000, E1   -72.940, E3 +86226.910}
SPL {X  -145.929, Y  +740.010, Z    +0.000, E1   -72.229, E3 +86243.382}
SPL {X  -139.114, Y  +753.439, Z    +0.000, E1   -71.436, E3 +86258.020}
SPL {X  -132.333, Y  +764.333, Z    +0.000, E1   -70.535, E3 +86270.644}
SPL {X  -125.486, Y  +773.664, Z    +0.000, E1   -69.598, E3 +86281.618}
SPL {X  -121.321, Y  +778.713, Z    +0.000, E1   -68.872, E3 +86287.628}
SPL {X   -77.337, Y  +814.468, Z    +0.000, E1   -56.377, E3 +86406.259}
ENDSPLINE

SPLINE
SPL {X  -134.727, Y  +760.706, Z    +0.000, E1   -50.460, E3 +86594.491}
SPL {X  -155.580, Y  +711.748, Z    +0.000, E1   -32.084, E3 +86611.406}
SPL {X  -159.445, Y  +687.715, Z    +0.000, E1   -14.660, E3 +86614.253}
SPL {X  -159.995, Y  +675.725, Z    +0.000, E1    -3.424, E3 +86614.764}
SPL {X  -160.000, Y  +671.714, Z    +0.000, E1    +0.835, E3 +86614.804}
SPL {X  -160.000, Y  +663.084, Z    +0.000, E1   +21.134, E3 +86615.128}
SPL {X  -160.000, Y  +650.910, Z    +0.000, E1   +46.005, E3 +86616.282}
SPL {X  -160.000, Y  +634.843, Z    +0.000, E1   +61.273, E3 +86618.959}
SPL {X  -160.000, Y  +578.679, Z    +0.000, E1   +71.665, E3 +86636.793}
SPL {X  -160.000, Y  +387.528, Z    +0.000, E1   +73.487, E3 +86729.605}
SPL {X  -159.218, Y  +369.903, Z    +0.000, E1   +73.425, E3 +86741.472}
SPL {X  -156.808, Y  +353.900, Z    +0.000, E1   +73.180, E3 +86754.076}
SPL {X  -154.539, Y  +344.254, Z    +0.000, E1   +72.827, E3 +86763.613}
ENDSPLINE

SPLINE
SPL {X  -157.258, Y  +356.206, Z    +0.000, E1   +70.434, E3 +86778.186}
ENDSPLINE

SPLINE
SPL {X  -150.342, Y  +330.952, Z    +0.000, E1   +71.154, E3 +86789.858}
SPL {X  -141.358, Y  +310.748, Z    +0.000, E1   +71.233, E3 +86802.564}
SPL {X  -134.330, Y  +298.778, Z    +0.000, E1   +70.323, E3 +86816.411}
SPL {X  -128.957, Y  +290.989, Z    +0.000, E1   +69.528, E3 +86825.776}
SPL {X  -124.846, Y  +285.632, Z    +0.000, E1   +68.906, E3 +86832.240}
SPL {X  -121.783, Y  +281.927, Z    +0.000, E1   +68.403, E3 +86836.672}
SPL {X   -79.219, Y  +246.688, Z    +0.000, E1   +55.887, E3 +86958.178}
ENDSPLINE

SPLINE
SPL {X  -125.038, Y  +285.873, Z    +0.000, E1   +53.023, E3 +87135.219}
SPL {X  -149.949, Y  +329.886, Z    +0.000, E1   +41.515, E3 +87156.784}
SPL {X  -157.246, Y  +356.141, Z    +0.000, E1   +27.282, E3 +87161.841}
SPL {X  -159.525, Y  +373.376, Z    +0.000, E1   +13.812, E3 +87163.498}
SPL {X  -160.000, Y  +387.264, Z    +0.000, E1    +0.544, E3 +87163.956}
SPL {X  -160.000, Y  +390.384, Z    +0.000, E1    -6.008, E3 +87163.993}
SPL {X  -160.000, Y  +395.752, Z    +0.000, E1   -19.038, E3 +87164.187}
SPL {X  -160.000, Y  +404.289, Z    +0.000, E1   -38.292, E3 +87164.855}
SPL {X  -160.000, Y  +418.681, Z    +0.000, E1   -56.949, E3 +87167.045}
SPL {X  -160.000, Y  +471.977, Z    +0.000, E1   -70.792, E3 +87183.564}
SPL {X  -159.977, Y  +677.138, Z    +0.000, E1   -73.665, E3 +87280.055}
SPL {X  -157.805, Y  +700.810, Z    +0.000, E1   -73.511, E3 +87296.885}
SPL {X  -152.242, Y  +723.618, Z    +0.000, E1   -72.940, E3 +87316.798}
SPL {X  -145.929, Y  +740.010, Z    +0.000, E1   -72.229, E3 +87333.270}
SPL {X  -139.114, Y  +753.439, Z    +0.000, E1   -71.436, E3 +87347.908}
SPL {X  -132.333, Y  +764.333, Z    +0.000, E1   -70.535, E3 +87360.532}
SPL {X  -125.486, Y  +773.664, Z    +0.000, E1   -69.598, E3 +87371.506}
SPL {X  -121.321, Y  +778.713, Z    +0.000, E1   -68.872, E3 +87377.516}
SPL {X   -77.337, Y  +814.468, Z    +0.000, E1   -56.377, E3 +87496.148}
ENDSPLINE

SPLINE
SPL {X  -134.727, Y  +760.706, Z    +0.000, E1   -50.460, E3 +87684.379}
SPL {X  -155.580, Y  +711.748, Z    +0.000, E1   -32.084, E3 +87701.294}
SPL {X  -159.445, Y  +687.715, Z    +0.000, E1   -14.660, E3 +87704.141}
SPL {X  -159.995, Y  +675.725, Z    +0.000, E1    -3.424, E3 +87704.652}
SPL {X  -160.000, Y  +671.714, Z    +0.000, E1    +0.835, E3 +87704.692}
SPL {X  -160.000, Y  +663.084, Z    +0.000, E1   +21.134, E3 +87705.016}
SPL {X  -160.000, Y  +650.910, Z    +0.000, E1   +46.005, E3 +87706.170}
SPL {X  -160.000, Y  +634.843, Z    +0.000, E1   +61.273, E3 +87708.847}
SPL {X  -160.000, Y  +578.679, Z    +0.000, E1   +71.665, E3 +87726.681}
SPL {X  -160.000, Y  +387.528, Z    +0.000, E1   +73.487, E3 +87819.493}
SPL {X  -159.218, Y  +369.903, Z    +0.000, E1   +73.425, E3 +87831.360}
SPL {X  -156.808, Y  +353.900, Z    +0.000, E1   +73.180, E3 +87843.964}
SPL {X  -154.539, Y  +344.254, Z    +0.000, E1   +72.827, E3 +87853.501}
ENDSPLINE

SPLINE
SPL {X  -157.258, Y  +356.206, Z    +0.000, E1   +70.434, E3 +87868.074}
ENDSPLINE

SPLINE
SPL {X  -150.342, Y  +330.952, Z    +0.000, E1   +71.154, E3 +87879.746}
SPL {X  -141.358, Y  +310.748, Z    +0.000, E1   +71.233, E3 +87892.452}
SPL {X  -134.330, Y  +298.778, Z    +0.000, E1   +70.323, E3 +87906.299}
SPL {X  -128.957, Y  +290.989, Z    +0.000, E1   +69.528, E3 +87915.664}
SPL {X  -124.846, Y  +285.632, Z    +0.000, E1   +68.906, E3 +87922.128}
SPL {X  -121.783, Y  +281.927, Z    +0.000, E1   +68.403, E3 +87926.560}
SPL {X   -79.219, Y  +246.688, Z    +0.000, E1   +55.887, E3 +88048.066}
ENDSPLINE

SPLINE
SPL {X  -125.038, Y  +285.873, Z    +0.000, E1   +53.023, E3 +88225.107}
SPL {X  -149.949, Y  +329.886, Z    +0.000, E1   +41.515, E3 +88246.672}
SPL {X  -157.246, Y  +356.141, Z    +0.000, E1   +27.282, E3 +88251.729}
SPL {X  -159.525, Y  +373.376, Z    +0.000, E1   +13.812, E3 +88253.386}
SPL {X  -160.000, Y  +387.264, Z    +0.000, E1    +0.544, E3 +88253.844}
SPL {X  -160.000, Y  +390.384, Z    +0.000, E1    -6.008, E3 +88253.881}
SPL {X  -160.000, Y  +395.752, Z    +0.000, E1   -19.038, E3 +88254.075}
SPL {X  -160.000, Y  +404.289, Z    +0.000, E1   -38.292, E3 +88254.743}
SPL {X  -160.000, Y  +418.681, Z    +0.000, E1   -56.949, E3 +88256.933}
SPL {X  -160.000, Y  +458.961, Z    +0.000, E1   -69.778, E3 +88268.529}
SPL {X  -160.000, Y  +485.343, Z    +0.000, E1   -71.539, E3 +88278.515}
SPL {X  -159.977, Y  +677.138, Z    +0.000, E1   -73.665, E3 +88369.943}
SPL {X  -157.805, Y  +700.810, Z    +0.000, E1   -73.511, E3 +88386.773}
SPL {X  -152.242, Y  +723.618, Z    +0.000, E1   -72.940, E3 +88406.686}
SPL {X  -145.929, Y  +740.010, Z    +0.000, E1   -72.229, E3 +88423.158}
SPL {X  -139.114, Y  +753.439, Z    +0.000, E1   -71.436, E3 +88437.796}
SPL {X  -132.333, Y  +764.333, Z    +0.000, E1   -70.535, E3 +88450.420}
SPL {X  -125.486, Y  +773.664, Z    +0.000, E1   -69.598, E3 +88461.394}
SPL {X  -121.321, Y  +778.713, Z    +0.000, E1   -68.872, E3 +88467.404}
SPL {X   -77.337, Y  +814.468, Z    +0.000, E1   -56.377, E3 +88586.036}
ENDSPLINE

SPLINE
SPL {X  -134.727, Y  +760.706, Z    +0.000, E1   -50.460, E3 +88774.267}
SPL {X  -155.580, Y  +711.748, Z    +0.000, E1   -32.084, E3 +88791.182}
SPL {X  -159.445, Y  +687.715, Z    +0.000, E1   -14.660, E3 +88794.029}
SPL {X  -159.995, Y  +675.725, Z    +0.000, E1    -3.424, E3 +88794.540}
SPL {X  -160.000, Y  +671.714, Z    +0.000, E1    +0.835, E3 +88794.580}
SPL {X  -160.000, Y  +663.084, Z    +0.000, E1   +21.134, E3 +88794.904}
SPL {X  -160.000, Y  +650.910, Z    +0.000, E1   +46.005, E3 +88796.058}
SPL {X  -160.000, Y  +634.843, Z    +0.000, E1   +61.273, E3 +88798.735}
SPL {X  -160.000, Y  +578.679, Z    +0.000, E1   +71.665, E3 +88816.569}
SPL {X  -160.000, Y  +387.528, Z    +0.000, E1   +73.487, E3 +88909.381}
SPL {X  -159.218, Y  +369.903, Z    +0.000, E1   +73.425, E3 +88921.248}
SPL {X  -156.808, Y  +353.900, Z    +0.000, E1   +73.180, E3 +88933.852}
SPL {X  -154.539, Y  +344.254, Z    +0.000, E1   +72.827, E3 +88943.389}
ENDSPLINE

SPLINE
SPL {X  -157.258, Y  +356.206, Z    +0.000, E1   +70.434, E3 +88957.962}
ENDSPLINE

SPLINE
SPL {X  -150.342, Y  +330.952, Z    +0.000, E1   +71.154, E3 +88969.634}
SPL {X  -141.358, Y  +310.748, Z    +0.000, E1   +71.233, E3 +88982.340}
SPL {X  -134.330, Y  +298.778, Z    +0.000, E1   +70.323, E3 +88996.187}
SPL {X  -128.957, Y  +290.989, Z    +0.000, E1   +69.528, E3 +89005.552}
SPL {X  -124.846, Y  +285.632, Z    +0.000, E1   +68.906, E3 +89012.016}
SPL {X  -121.783, Y  +281.927, Z    +0.000, E1   +68.403, E3 +89016.448}
SPL {X   -79.219, Y  +246.688, Z    +0.000, E1   +55.887, E3 +89137.954}
ENDSPLINE

SPLINE
SPL {X  -125.038, Y  +285.873, Z    +0.000, E1   +53.023, E3 +89314.995}
SPL {X  -149.949, Y  +329.886, Z    +0.000, E1   +41.515, E3 +89336.560}
SPL {X  -157.246, Y  +356.141, Z    +0.000, E1   +27.282, E3 +89341.617}
SPL {X  -159.525, Y  +373.376, Z    +0.000, E1   +13.812, E3 +89343.274}
SPL {X  -160.000, Y  +387.264, Z    +0.000, E1    +0.544, E3 +89343.732}
SPL {X  -160.000, Y  +390.384, Z    +0.000, E1    -6.008, E3 +89343.769}
SPL {X  -160.000, Y  +395.752, Z    +0.000, E1   -19.038, E3 +89343.963}
SPL {X  -160.000, Y  +404.289, Z    +0.000, E1   -38.292, E3 +89344.631}
SPL {X  -160.000, Y  +418.681, Z    +0.000, E1   -56.949, E3 +89346.821}
SPL {X  -160.000, Y  +471.977, Z    +0.000, E1   -70.792, E3 +89363.340}
SPL {X  -159.977, Y  +677.138, Z    +0.000, E1   -73.665, E3 +89459.831}
SPL {X  -157.805, Y  +700.810, Z    +0.000, E1   -73.511, E3 +89476.662}
SPL {X  -152.242, Y  +723.618, Z    +0.000, E1   -72.940, E3 +89496.574}
SPL {X  -145.929, Y  +740.010, Z    +0.000, E1   -72.229, E3 +89513.046}
SPL {X  -139.114, Y  +753.439, Z    +0.000, E1   -71.436, E3 +89527.684}
SPL {X  -132.333, Y  +764.333, Z    +0.000, E1   -70.535, E3 +89540.308}
SPL {X  -125.486, Y  +773.664, Z    +0.000, E1   -69.598, E3 +89551.282}
SPL {X  -121.321, Y  +778.713, Z    +0.000, E1   -68.872, E3 +89557.292}
SPL {X   -77.337, Y  +814.468, Z    +0.000, E1   -56.377, E3 +89675.924}
ENDSPLINE

SPLINE
SPL {X  -134.727, Y  +760.706, Z    +0.000, E1   -50.460, E3 +89864.155}
SPL {X  -155.580, Y  +711.748, Z    +0.000, E1   -32.084, E3 +89881.070}
SPL {X  -159.445, Y  +687.715, Z    +0.000, E1   -14.660, E3 +89883.917}
SPL {X  -159.995, Y  +675.725, Z    +0.000, E1    -3.424, E3 +89884.428}
SPL {X  -160.000, Y  +671.714, Z    +0.000, E1    +0.835, E3 +89884.468}
SPL {X  -160.000, Y  +663.084, Z    +0.000, E1   +21.134, E3 +89884.792}
SPL {X  -160.000, Y  +650.910, Z    +0.000, E1   +46.005, E3 +89885.946}
SPL {X  -160.000, Y  +634.843, Z    +0.000, E1   +61.273, E3 +89888.623}
SPL {X  -160.000, Y  +578.679, Z    +0.000, E1   +71.665, E3 +89906.457}
SPL {X  -160.000, Y  +387.528, Z    +0.000, E1   +73.487, E3 +89999.269}
SPL {X  -159.218, Y  +369.903, Z    +0.000, E1   +73.425, E3 +90011.136}
SPL {X  -156.808, Y  +353.900, Z    +0.000, E1   +73.180, E3 +90023.740}
SPL {X  -154.539, Y  +344.254, Z    +0.000, E1   +72.827, E3 +90033.278}
ENDSPLINE

SPLINE
SPL {X  -157.258, Y  +356.206, Z    +0.000, E1   +70.434, E3 +90047.850}
ENDSPLINE

SPLINE
SPL {X  -150.342, Y  +330.952, Z    +0.000, E1   +71.154, E3 +90059.522}
SPL {X  -141.358, Y  +310.748, Z    +0.000, E1   +71.233, E3 +90072.228}
SPL {X  -134.330, Y  +298.778, Z    +0.000, E1   +70.323, E3 +90086.075}
SPL {X  -128.957, Y  +290.989, Z    +0.000, E1   +69.528, E3 +90095.440}
SPL {X  -124.846, Y  +285.632, Z    +0.000, E1   +68.906, E3 +90101.904}
SPL {X  -121.783, Y  +281.927, Z    +0.000, E1   +68.403, E3 +90106.336}
SPL {X   -79.219, Y  +246.688, Z    +0.000, E1   +55.887, E3 +90227.842}
ENDSPLINE

SPLINE
SPL {X  -125.038, Y  +285.873, Z    +0.000, E1   +53.023, E3 +90404.883}
SPL {X  -149.949, Y  +329.886, Z    +0.000, E1   +41.515, E3 +90426.448}
SPL {X  -157.246, Y  +356.141, Z    +0.000, E1   +27.282, E3 +90431.505}
SPL {X  -159.525, Y  +373.376, Z    +0.000, E1   +13.812, E3 +90433.162}
SPL {X  -160.000, Y  +387.264, Z    +0.000, E1    +0.544, E3 +90433.620}
SPL {X  -160.000, Y  +390.384, Z    +0.000, E1    -6.008, E3 +90433.657}
SPL {X  -160.000, Y  +395.752, Z    +0.000, E1   -19.038, E3 +90433.851}
SPL {X  -160.000, Y  +404.289, Z    +0.000, E1   -38.292, E3 +90434.519}
SPL {X  -160.000, Y  +418.681, Z    +0.000, E1   -56.949, E3 +90436.709}
SPL {X  -160.000, Y  +471.977, Z    +0.000, E1   -70.792, E3 +90453.228}
SPL {X  -159.977, Y  +677.138, Z    +0.000, E1   -73.665, E3 +90549.719}
SPL {X  -157.805, Y  +700.810, Z    +0.000, E1   -73.511, E3 +90566.550}
SPL {X  -152.242, Y  +723.618, Z    +0.000, E1   -72.940, E3 +90586.462}
SPL {X  -145.929, Y  +740.010, Z    +0.000, E1   -72.229, E3 +90602.934}
SPL {X  -139.114, Y  +753.439, Z    +0.000, E1   -71.436, E3 +90617.572}
SPL {X  -132.333, Y  +764.333, Z    +0.000, E1   -70.535, E3 +90630.196}
SPL {X  -125.486, Y  +773.664, Z    +0.000, E1   -69.598, E3 +90641.170}
SPL {X  -121.321, Y  +778.713, Z    +0.000, E1   -68.872, E3 +90647.180}
SPL {X   -77.337, Y  +814.468, Z    +0.000, E1   -56.377, E3 +90765.812}
ENDSPLINE

SPLINE
SPL {X  -134.727, Y  +760.706, Z    +0.000, E1   -50.460, E3 +90954.044}
SPL {X  -155.580, Y  +711.748, Z    +0.000, E1   -32.084, E3 +90970.958}
SPL {X  -159.445, Y  +687.715, Z    +0.000, E1   -14.660, E3 +90973.805}
SPL {X  -159.995, Y  +675.725, Z    +0.000, E1    -3.424, E3 +90974.316}
SPL {X  -160.000, Y  +671.714, Z    +0.000, E1    +0.835, E3 +90974.356}
SPL {X  -160.000, Y  +663.084, Z    +0.000, E1   +21.134, E3 +90974.681}
SPL {X  -160.000, Y  +650.910, Z    +0.000, E1   +46.005, E3 +90975.834}
SPL {X  -160.000, Y  +634.843, Z    +0.000, E1   +61.273, E3 +90978.511}
SPL {X  -160.000, Y  +578.679, Z    +0.000, E1   +71.665, E3 +90996.345}
SPL {X  -160.000, Y  +387.528, Z    +0.000, E1   +73.487, E3 +91089.157}
SPL {X  -159.218, Y  +369.903, Z    +0.000, E1   +73.425, E3 +91101.024}
SPL {X  -156.808, Y  +353.900, Z    +0.000, E1   +73.180, E3 +91113.628}
SPL {X  -154.539, Y  +344.254, Z    +0.000, E1   +72.827, E3 +91123.166}
ENDSPLINE

SPLINE
SPL {X  -157.258, Y  +356.206, Z    +0.000, E1   +70.434, E3 +91137.738}
ENDSPLINE

SPLINE
SPL {X  -150.342, Y  +330.952, Z    +0.000, E1   +71.154, E3 +91149.410}
SPL {X  -141.358, Y  +310.748, Z    +0.000, E1   +71.233, E3 +91162.116}
SPL {X  -134.330, Y  +298.778, Z    +0.000, E1   +70.323, E3 +91175.963}
SPL {X  -128.957, Y  +290.989, Z    +0.000, E1   +69.528, E3 +91185.329}
SPL {X  -124.846, Y  +285.632, Z    +0.000, E1   +68.906, E3 +91191.792}
SPL {X  -121.783, Y  +281.927, Z    +0.000, E1   +68.403, E3 +91196.224}
SPL {X   -79.219, Y  +246.688, Z    +0.000, E1   +55.887, E3 +91317.730}
ENDSPLINE

SPLINE
SPL {X  -125.038, Y  +285.873, Z    +0.000, E1   +53.023, E3 +91494.771}
SPL {X  -149.949, Y  +329.886, Z    +0.000, E1   +41.515, E3 +91516.337}
SPL {X  -157.246, Y  +356.141, Z    +0.000, E1   +27.282, E3 +91521.393}
SPL {X  -159.525, Y  +373.376, Z    +0.000, E1   +13.812, E3 +91523.050}
SPL {X  -160.000, Y  +387.264, Z    +0.000, E1    +0.544, E3 +91523.508}
SPL {X  -160.000, Y  +390.384, Z    +0.000, E1    -6.008, E3 +91523.545}
SPL {X  -160.000, Y  +395.752, Z    +0.000, E1   -19.038, E3 +91523.739}
SPL {X  -160.000, Y  +404.289, Z    +0.000, E1   -38.292, E3 +91524.407}
SPL {X  -160.000, Y  +418.681, Z    +0.000, E1   -56.949, E3 +91526.597}
SPL {X  -160.000, Y  +471.977, Z    +0.000, E1   -70.792, E3 +91543.116}
SPL {X  -159.977, Y  +677.138, Z    +0.000, E1   -73.665, E3 +91639.607}
SPL {X  -157.805, Y  +700.810, Z    +0.000, E1   -73.511, E3 +91656.438}
SPL {X  -152.242, Y  +723.618, Z    +0.000, E1   -72.940, E3 +91676.350}
SPL {X  -145.929, Y  +740.010, Z    +0.000, E1   -72.229, E3 +91692.822}
SPL {X  -139.114, Y  +753.439, Z    +0.000, E1   -71.436, E3 +91707.460}
SPL {X  -132.333, Y  +764.333, Z    +0.000, E1   -70.535, E3 +91720.084}
SPL {X  -125.486, Y  +773.664, Z    +0.000, E1   -69.598, E3 +91731.058}
SPL {X  -121.321, Y  +778.713, Z    +0.000, E1   -68.872, E3 +91737.068}
SPL {X   -77.337, Y  +814.468, Z    +0.000, E1   -56.377, E3 +91855.700}
ENDSPLINE

SPLINE
SPL {X  -134.727, Y  +760.706, Z    +0.000, E1   -50.460, E3 +92043.932}
SPL {X  -155.580, Y  +711.748, Z    +0.000, E1   -32.084, E3 +92060.846}
SPL {X  -159.445, Y  +687.715, Z    +0.000, E1   -14.660, E3 +92063.693}
SPL {X  -159.995, Y  +675.725, Z    +0.000, E1    -3.424, E3 +92064.204}
SPL {X  -160.000, Y  +671.714, Z    +0.000, E1    +0.835, E3 +92064.244}
SPL {X  -160.000, Y  +663.084, Z    +0.000, E1   +21.134, E3 +92064.569}
SPL {X  -160.000, Y  +650.910, Z    +0.000, E1   +46.005, E3 +92065.722}
SPL {X  -160.000, Y  +634.843, Z    +0.000, E1   +61.273, E3 +92068.399}
SPL {X  -160.000, Y  +578.679, Z    +0.000, E1   +71.665, E3 +92086.233}
SPL {X  -160.000, Y  +387.528, Z    +0.000, E1   +73.487, E3 +92179.045}
SPL {X  -159.218, Y  +369.903, Z    +0.000, E1   +73.425, E3 +92190.913}
SPL {X  -156.808, Y  +353.900, Z    +0.000, E1   +73.180, E3 +92203.516}
SPL {X  -154.539, Y  +344.254, Z    +0.000, E1   +72.827, E3 +92213.054}
ENDSPLINE

SPLINE
SPL {X  -157.258, Y  +356.206, Z    +0.000, E1   +70.434, E3 +92227.626}
ENDSPLINE

SPLINE
SPL {X  -150.342, Y  +330.952, Z    +0.000, E1   +71.154, E3 +92239.298}
SPL {X  -141.358, Y  +310.748, Z    +0.000, E1   +71.233, E3 +92252.004}
SPL {X  -134.330, Y  +298.778, Z    +0.000, E1   +70.323, E3 +92265.851}
SPL {X  -128.957, Y  +290.989, Z    +0.000, E1   +69.528, E3 +92275.217}
SPL {X  -124.846, Y  +285.632, Z    +0.000, E1   +68.906, E3 +92281.680}
SPL {X  -121.783, Y  +281.927, Z    +0.000, E1   +68.403, E3 +92286.112}
SPL {X   -79.219, Y  +246.688, Z    +0.000, E1   +55.887, E3 +92407.618}
ENDSPLINE

SPLINE
SPL {X  -125.038, Y  +285.873, Z    +0.000, E1   +53.023, E3 +92584.660}
SPL {X  -149.949, Y  +329.886, Z    +0.000, E1   +41.515, E3 +92606.225}
SPL {X  -157.246, Y  +356.141, Z    +0.000, E1   +27.282, E3 +92611.281}
SPL {X  -159.525, Y  +373.376, Z    +0.000, E1   +13.812, E3 +92612.938}
SPL {X  -160.000, Y  +387.264, Z    +0.000, E1    +0.544, E3 +92613.396}
SPL {X  -160.000, Y  +390.384, Z    +0.000, E1    -6.008, E3 +92613.433}
SPL {X  -160.000, Y  +395.752, Z    +0.000, E1   -19.038, E3 +92613.627}
SPL {X  -160.000, Y  +404.289, Z    +0.000, E1   -38.292, E3 +92614.295}
SPL {X  -160.000, Y  +418.681, Z    +0.000, E1   -56.949, E3 +92616.485}
SPL {X  -160.000, Y  +471.977, Z    +0.000, E1   -70.792, E3 +92633.004}
SPL {X  -159.977, Y  +677.138, Z    +0.000, E1   -73.665, E3 +92729.495}
SPL {X  -157.805, Y  +700.810, Z    +0.000, E1   -73.511, E3 +92746.326}
SPL {X  -152.242, Y  +723.618, Z    +0.000, E1   -72.940, E3 +92766.239}
SPL {X  -145.929, Y  +740.010, Z    +0.000, E1   -72.229, E3 +92782.710}
SPL {X  -139.114, Y  +753.439, Z    +0.000, E1   -71.436, E3 +92797.349}
SPL {X  -132.333, Y  +764.333, Z    +0.000, E1   -70.535, E3 +92809.972}
SPL {X  -125.486, Y  +773.664, Z    +0.000, E1   -69.598, E3 +92820.947}
SPL {X  -121.321, Y  +778.713, Z    +0.000, E1   -68.872, E3 +92826.957}
SPL {X   -77.337, Y  +814.468, Z    +0.000, E1   -56.377, E3 +92945.588}
ENDSPLINE

SPLINE
SPL {X  -134.727, Y  +760.706, Z    +0.000, E1   -50.460, E3 +93133.820}
SPL {X  -155.580, Y  +711.748, Z    +0.000, E1   -32.084, E3 +93150.734}
SPL {X  -159.445, Y  +687.715, Z    +0.000, E1   -14.660, E3 +93153.581}
SPL {X  -159.995, Y  +675.725, Z    +0.000, E1    -3.424, E3 +93154.092}
SPL {X  -160.000, Y  +671.714, Z    +0.000, E1    +0.835, E3 +93154.132}
SPL {X  -160.000, Y  +663.084, Z    +0.000, E1   +21.134, E3 +93154.457}
SPL {X  -160.000, Y  +650.910, Z    +0.000, E1   +46.005, E3 +93155.610}
SPL {X  -160.000, Y  +634.843, Z    +0.000, E1   +61.273, E3 +93158.287}
SPL {X  -160.000, Y  +578.679, Z    +0.000, E1   +71.665, E3 +93176.121}
SPL {X  -160.000, Y  +387.528, Z    +0.000, E1   +73.487, E3 +93268.933}
SPL {X  -159.218, Y  +369.903, Z    +0.000, E1   +73.425, E3 +93280.801}
SPL {X  -156.808, Y  +353.900, Z    +0.000, E1   +73.180, E3 +93293.404}
SPL {X  -154.539, Y  +344.254, Z    +0.000, E1   +72.827, E3 +93302.942}
ENDSPLINE

SPLINE
SPL {X  -157.258, Y  +356.206, Z    +0.000, E1   +70.434, E3 +93317.514}
ENDSPLINE

SPLINE
SPL {X  -150.342, Y  +330.952, Z    +0.000, E1   +71.154, E3 +93329.186}
SPL {X  -141.358, Y  +310.748, Z    +0.000, E1   +71.233, E3 +93341.892}
SPL {X  -134.330, Y  +298.778, Z    +0.000, E1   +70.323, E3 +93355.739}
SPL {X  -128.957, Y  +290.989, Z    +0.000, E1   +69.528, E3 +93365.105}
SPL {X  -124.846, Y  +285.632, Z    +0.000, E1   +68.906, E3 +93371.568}
SPL {X  -121.783, Y  +281.927, Z    +0.000, E1   +68.403, E3 +93376.000}
SPL {X   -79.219, Y  +246.688, Z    +0.000, E1   +55.887, E3 +93497.506}
ENDSPLINE

SPLINE
SPL {X  -125.038, Y  +285.873, Z    +0.000, E1   +53.023, E3 +93674.548}
SPL {X  -149.949, Y  +329.886, Z    +0.000, E1   +41.515, E3 +93696.113}
SPL {X  -157.246, Y  +356.141, Z    +0.000, E1   +27.282, E3 +93701.169}
SPL {X  -159.525, Y  +373.376, Z    +0.000, E1   +13.812, E3 +93702.826}
SPL {X  -160.000, Y  +387.264, Z    +0.000, E1    +0.544, E3 +93703.284}
SPL {X  -160.000, Y  +390.384, Z    +0.000, E1    -6.008, E3 +93703.321}
SPL {X  -160.000, Y  +395.752, Z    +0.000, E1   -19.038, E3 +93703.515}
SPL {X  -160.000, Y  +404.289, Z    +0.000, E1   -38.292, E3 +93704.183}
SPL {X  -160.000, Y  +418.681, Z    +0.000, E1   -56.949, E3 +93706.373}
SPL {X  -160.000, Y  +471.977, Z    +0.000, E1   -70.792, E3 +93722.892}
SPL {X  -159.977, Y  +677.138, Z    +0.000, E1   -73.665, E3 +93819.383}
SPL {X  -157.805, Y  +700.810, Z    +0.000, E1   -73.511, E3 +93836.214}
SPL {X  -152.242, Y  +723.618, Z    +0.000, E1   -72.940, E3 +93856.127}
SPL {X  -145.929, Y  +740.010, Z    +0.000, E1   -72.229, E3 +93872.598}
SPL {X  -139.114, Y  +753.439, Z    +0.000, E1   -71.436, E3 +93887.237}
SPL {X  -132.333, Y  +764.333, Z    +0.000, E1   -70.535, E3 +93899.860}
SPL {X  -125.486, Y  +773.664, Z    +0.000, E1   -69.598, E3 +93910.835}
SPL {X  -121.321, Y  +778.713, Z    +0.000, E1   -68.872, E3 +93916.845}
SPL {X   -77.337, Y  +814.468, Z    +0.000, E1   -56.377, E3 +94035.476}
ENDSPLINE

SPLINE
SPL {X  -134.727, Y  +760.706, Z    +0.000, E1   -50.460, E3 +94223.708}
SPL {X  -155.580, Y  +711.748, Z    +0.000, E1   -32.084, E3 +94240.622}
SPL {X  -159.445, Y  +687.715, Z    +0.000, E1   -14.660, E3 +94243.469}
SPL {X  -159.995, Y  +675.725, Z    +0.000, E1    -3.424, E3 +94243.980}
SPL {X  -160.000, Y  +671.714, Z    +0.000, E1    +0.835, E3 +94244.020}
SPL {X  -160.000, Y  +663.084, Z    +0.000, E1   +21.134, E3 +94244.345}
SPL {X  -160.000, Y  +650.910, Z    +0.000, E1   +46.005, E3 +94245.498}
SPL {X  -160.000, Y  +634.843, Z    +0.000, E1   +61.273, E3 +94248.175}
SPL {X  -160.000, Y  +578.679, Z    +0.000, E1   +71.665, E3 +94266.009}
SPL {X  -160.000, Y  +387.528, Z    +0.000, E1   +73.487, E3 +94358.821}
SPL {X  -159.218, Y  +369.903, Z    +0.000, E1   +73.425, E3 +94370.689}
SPL {X  -156.808, Y  +353.900, Z    +0.000, E1   +73.180, E3 +94383.292}
SPL {X  -154.539, Y  +344.254, Z    +0.000, E1   +72.827, E3 +94392.830}
ENDSPLINE

SPLINE
SPL {X  -157.258, Y  +356.206, Z    +0.000, E1   +70.434, E3 +94407.402}
ENDSPLINE

SPLINE
SPL {X  -150.342, Y  +330.952, Z    +0.000, E1   +71.154, E3 +94419.074}
SPL {X  -141.358, Y  +310.748, Z    +0.000, E1   +71.233, E3 +94431.780}
SPL {X  -134.330, Y  +298.778, Z    +0.000, E1   +70.323, E3 +94445.627}
SPL {X  -128.957, Y  +290.989, Z    +0.000, E1   +69.528, E3 +94454.993}
SPL {X  -124.846, Y  +285.632, Z    +0.000, E1   +68.906, E3 +94461.456}
SPL {X  -121.783, Y  +281.927, Z    +0.000, E1   +68.403, E3 +94465.888}
SPL {X   -79.219, Y  +246.688, Z    +0.000, E1   +55.887, E3 +94587.394}
ENDSPLINE

SPLINE
SPL {X  -125.038, Y  +285.873, Z    +0.000, E1   +53.023, E3 +94764.436}
SPL {X  -149.949, Y  +329.886, Z    +0.000, E1   +41.515, E3 +94786.001}
SPL {X  -157.246, Y  +356.141, Z    +0.000, E1   +27.282, E3 +94791.057}
SPL {X  -159.525, Y  +373.376, Z    +0.000, E1   +13.812, E3 +94792.714}
SPL {X  -160.000, Y  +387.264, Z    +0.000, E1    +0.544, E3 +94793.172}
SPL {X  -160.000, Y  +390.384, Z    +0.000, E1    -6.008, E3 +94793.209}
SPL {X  -160.000, Y  +395.752, Z    +0.000, E1   -19.038, E3 +94793.403}
SPL {X  -160.000, Y  +404.289, Z    +0.000, E1   -38.292, E3 +94794.071}
SPL {X  -160.000, Y  +418.681, Z    +0.000, E1   -56.949, E3 +94796.261}
SPL {X  -160.000, Y  +471.977, Z    +0.000, E1   -70.792, E3 +94812.780}
SPL {X  -159.977, Y  +677.138, Z    +0.000, E1   -73.665, E3 +94909.271}
SPL {X  -157.805, Y  +700.810, Z    +0.000, E1   -73.511, E3 +94926.102}
SPL {X  -152.242, Y  +723.618, Z    +0.000, E1   -72.940, E3 +94946.015}
SPL {X  -145.929, Y  +740.010, Z    +0.000, E1   -72.229, E3 +94962.486}
SPL {X  -139.114, Y  +753.439, Z    +0.000, E1   -71.436, E3 +94977.125}
SPL {X  -132.333, Y  +764.333, Z    +0.000, E1   -70.535, E3 +94989.748}
SPL {X  -125.486, Y  +773.664, Z    +0.000, E1   -69.598, E3 +95000.723}
SPL {X  -121.321, Y  +778.713, Z    +0.000, E1   -68.872, E3 +95006.733}
SPL {X   -77.337, Y  +814.468, Z    +0.000, E1   -56.377, E3 +95125.364}
ENDSPLINE

SPLINE
SPL {X  -134.727, Y  +760.706, Z    +0.000, E1   -50.460, E3 +95313.596}
SPL {X  -155.580, Y  +711.748, Z    +0.000, E1   -32.084, E3 +95330.510}
SPL {X  -159.445, Y  +687.715, Z    +0.000, E1   -14.660, E3 +95333.357}
SPL {X  -159.995, Y  +675.725, Z    +0.000, E1    -3.424, E3 +95333.868}
SPL {X  -160.000, Y  +671.714, Z    +0.000, E1    +0.835, E3 +95333.908}
SPL {X  -160.000, Y  +663.084, Z    +0.000, E1   +21.134, E3 +95334.233}
SPL {X  -160.000, Y  +650.910, Z    +0.000, E1   +46.005, E3 +95335.386}
SPL {X  -160.000, Y  +634.843, Z    +0.000, E1   +61.273, E3 +95338.063}
SPL {X  -160.000, Y  +578.679, Z    +0.000, E1   +71.665, E3 +95355.897}
SPL {X  -160.000, Y  +387.528, Z    +0.000, E1   +73.487, E3 +95448.709}
SPL {X  -159.218, Y  +369.903, Z    +0.000, E1   +73.425, E3 +95460.577}
SPL {X  -156.808, Y  +353.900, Z    +0.000, E1   +73.180, E3 +95473.180}
SPL {X  -154.539, Y  +344.254, Z    +0.000, E1   +72.827, E3 +95482.718}
ENDSPLINE

SPLINE
SPL {X  -157.258, Y  +356.206, Z    +0.000, E1   +70.434, E3 +95497.290}
ENDSPLINE

SPLINE
SPL {X  -150.342, Y  +330.952, Z    +0.000, E1   +71.154, E3 +95508.962}
SPL {X  -141.358, Y  +310.748, Z    +0.000, E1   +71.233, E3 +95521.668}
SPL {X  -134.330, Y  +298.778, Z    +0.000, E1   +70.323, E3 +95535.515}
SPL {X  -128.957, Y  +290.989, Z    +0.000, E1   +69.528, E3 +95544.881}
SPL {X  -124.846, Y  +285.632, Z    +0.000, E1   +68.906, E3 +95551.344}
SPL {X  -121.783, Y  +281.927, Z    +0.000, E1   +68.403, E3 +95555.776}
SPL {X   -79.219, Y  +246.688, Z    +0.000, E1   +55.887, E3 +95677.282}
ENDSPLINE

SPLINE
SPL {X  -125.038, Y  +285.873, Z    +0.000, E1   +53.023, E3 +95854.324}
SPL {X  -149.949, Y  +329.886, Z    +0.000, E1   +41.515, E3 +95875.889}
SPL {X  -157.246, Y  +356.141, Z    +0.000, E1   +27.282, E3 +95880.945}
SPL {X  -159.525, Y  +373.376, Z    +0.000, E1   +13.812, E3 +95882.602}
SPL {X  -160.000, Y  +387.264, Z    +0.000, E1    +0.544, E3 +95883.060}
SPL {X  -160.000, Y  +390.384, Z    +0.000, E1    -6.008, E3 +95883.097}
SPL {X  -160.000, Y  +395.752, Z    +0.000, E1   -19.038, E3 +95883.291}
SPL {X  -160.000, Y  +404.289, Z    +0.000, E1   -38.292, E3 +95883.959}
SPL {X  -160.000, Y  +418.681, Z    +0.000, E1   -56.949, E3 +95886.149}
SPL {X  -160.000, Y  +471.977, Z    +0.000, E1   -70.792, E3 +95902.668}
SPL {X  -159.977, Y  +677.138, Z    +0.000, E1   -73.665, E3 +95999.160}
SPL {X  -157.805, Y  +700.810, Z    +0.000, E1   -73.511, E3 +96015.990}
SPL {X  -152.242, Y  +723.618, Z    +0.000, E1   -72.940, E3 +96035.903}
SPL {X  -145.929, Y  +740.010, Z    +0.000, E1   -72.229, E3 +96052.374}
SPL {X  -139.114, Y  +753.439, Z    +0.000, E1   -71.436, E3 +96067.013}
SPL {X  -132.333, Y  +764.333, Z    +0.000, E1   -70.535, E3 +96079.636}
SPL {X  -125.486, Y  +773.664, Z    +0.000, E1   -69.598, E3 +96090.611}
SPL {X  -121.321, Y  +778.713, Z    +0.000, E1   -68.872, E3 +96096.621}
SPL {X   -77.337, Y  +814.468, Z    +0.000, E1   -56.377, E3 +96215.252}
ENDSPLINE

SPLINE
SPL {X  -134.727, Y  +760.706, Z    +0.000, E1   -50.460, E3 +96403.484}
SPL {X  -155.580, Y  +711.748, Z    +0.000, E1   -32.084, E3 +96420.398}
SPL {X  -159.445, Y  +687.715, Z    +0.000, E1   -14.660, E3 +96423.245}
SPL {X  -159.995, Y  +675.725, Z    +0.000, E1    -3.424, E3 +96423.756}
SPL {X  -160.000, Y  +671.714, Z    +0.000, E1    +0.835, E3 +96423.796}
SPL {X  -160.000, Y  +663.084, Z    +0.000, E1   +21.134, E3 +96424.121}
SPL {X  -160.000, Y  +650.910, Z    +0.000, E1   +46.005, E3 +96425.274}
SPL {X  -160.000, Y  +634.843, Z    +0.000, E1   +61.273, E3 +96427.951}
SPL {X  -160.000, Y  +578.679, Z    +0.000, E1   +71.665, E3 +96445.785}
SPL {X  -160.000, Y  +387.528, Z    +0.000, E1   +73.487, E3 +96538.597}
SPL {X  -159.218, Y  +369.903, Z    +0.000, E1   +73.425, E3 +96550.465}
SPL {X  -156.808, Y  +353.900, Z    +0.000, E1   +73.180, E3 +96563.068}
SPL {X  -154.539, Y  +344.254, Z    +0.000, E1   +72.827, E3 +96572.606}
ENDSPLINE

SPLINE
SPL {X  -157.258, Y  +356.206, Z    +0.000, E1   +70.434, E3 +96587.178}
ENDSPLINE

SPLINE
SPL {X  -150.342, Y  +330.952, Z    +0.000, E1   +71.154, E3 +96598.851}
ENDSPLINE

SPLINE
SPL {X  -147.383, Y  +323.425, Z    +0.000, E1   +69.849, E3 +96614.426}
SPL {X  -143.458, Y  +314.849, Z    +0.000, E1   +69.330, E3 +96624.353}
SPL {X  -137.919, Y  +304.592, Z    +0.000, E1   +68.645, E3 +96636.642}
SPL {X  -132.252, Y  +295.648, Z    +0.000, E1   +67.759, E3 +96647.957}
SPL {X  -127.852, Y  +289.504, Z    +0.000, E1   +67.080, E3 +96655.789}
SPL {X  -124.264, Y  +284.911, Z    +0.000, E1   +66.468, E3 +96661.685}
SPL {X   -87.531, Y  +251.766, Z    +0.000, E1   +54.242, E3 +96790.001}
ENDSPLINE

SPLINE
SPL {X  -130.414, Y  +293.006, Z    +0.000, E1   +48.816, E3 +96938.614}
SPL {X  -151.093, Y  +333.061, Z    +0.000, E1   +36.955, E3 +96959.894}
SPL {X  -158.896, Y  +366.939, Z    +0.000, E1   +17.535, E3 +96966.434}
SPL {X  -160.000, Y  +387.267, Z    +0.000, E1    +0.577, E3 +96967.624}
SPL {X  -160.000, Y  +391.471, Z    +0.000, E1    -7.208, E3 +96967.705}
SPL {X  -160.000, Y  +398.523, Z    +0.000, E1   -22.265, E3 +96968.117}
SPL {X  -160.000, Y  +411.325, Z    +0.000, E1   -44.857, E3 +96969.783}
SPL {X  -160.000, Y  +459.786, Z    +0.000, E1   -66.828, E3 +96985.175}
SPL {X  -160.000, Y  +650.407, Z    +0.000, E1   -71.387, E3 +97087.832}
SPL {X  -159.770, Y  +682.971, Z    +0.000, E1   -71.362, E3 +97111.408}
SPL {X  -156.288, Y  +708.665, Z    +0.000, E1   -70.996, E3 +97133.418}
SPL {X  -150.837, Y  +727.770, Z    +0.000, E1   -70.337, E3 +97152.752}
SPL {X  -144.661, Y  +742.760, Z    +0.000, E1   -69.570, E3 +97169.510}
SPL {X  -137.606, Y  +756.037, Z    +0.000, E1   -68.631, E3 +97185.475}
SPL {X  -131.907, Y  +764.957, Z    +0.000, E1   -67.736, E3 +97196.770}
SPL {X  -127.608, Y  +770.921, Z    +0.000, E1   -67.067, E3 +97204.388}
SPL {X  -124.072, Y  +775.426, Z    +0.000, E1   -66.459, E3 +97210.169}
SPL {X   -86.375, Y  +809.082, Z    +0.000, E1   -54.606, E3 +97334.499}
ENDSPLINE

SPLINE
SPL {X  -131.819, Y  +765.085, Z    +0.000, E1   -48.689, E3 +97490.392}
SPL {X  -153.047, Y  +721.053, Z    +0.000, E1   -34.410, E3 +97510.258}
SPL {X  -159.196, Y  +690.423, Z    +0.000, E1   -15.522, E3 +97515.355}
SPL {X  -160.000, Y  +672.957, Z    +0.000, E1    -0.766, E3 +97516.257}
SPL {X  -160.000, Y  +670.573, Z    +0.000, E1    +3.229, E3 +97516.285}
SPL {X  -160.000, Y  +665.683, Z    +0.000, E1   +13.339, E3 +97516.454}
SPL {X  -160.000, Y  +658.186, Z    +0.000, E1   +29.314, E3 +97517.058}
SPL {X  -160.000, Y  +642.169, Z    +0.000, E1   +52.097, E3 +97519.584}
SPL {X  -160.000, Y  +581.106, Z    +0.000, E1   +69.111, E3 +97540.456}
SPL {X  -160.000, Y  +418.281, Z    +0.000, E1   +71.209, E3 +97631.806}
SPL {X  -153.877, Y  +341.861, Z    +0.000, E1   +74.632, E3 +97645.219}
SPL {X  -152.649, Y  +337.758, Z    +0.000, E1   +72.728, E3 +97666.882}
SPL {X  -150.568, Y  +331.578, Z    +0.000, E1   +70.963, E3 +97686.808}
SPL {X  -147.367, Y  +323.387, Z    +0.000, E1   +69.846, E3 +97701.428}
SPL {X  -143.458, Y  +314.849, Z    +0.000, E1   +69.330, E3 +97711.310}
SPL {X  -137.919, Y  +304.592, Z    +0.000, E1   +68.645, E3 +97723.599}
SPL {X  -132.252, Y  +295.648, Z    +0.000, E1   +67.759, E3 +97734.914}
SPL {X  -127.852, Y  +289.504, Z    +0.000, E1   +67.080, E3 +97742.746}
SPL {X  -124.264, Y  +284.911, Z    +0.000, E1   +66.468, E3 +97748.642}
SPL {X   -87.531, Y  +251.766, Z    +0.000, E1   +54.242, E3 +97876.959}
ENDSPLINE

SPLINE
SPL {X  -130.414, Y  +293.006, Z    +0.000, E1   +48.816, E3 +98025.571}
SPL {X  -151.093, Y  +333.061, Z    +0.000, E1   +36.955, E3 +98046.852}
SPL {X  -158.896, Y  +366.939, Z    +0.000, E1   +17.535, E3 +98053.391}
SPL {X  -160.000, Y  +387.267, Z    +0.000, E1    +0.577, E3 +98054.581}
SPL {X  -160.000, Y  +391.471, Z    +0.000, E1    -7.208, E3 +98054.662}
SPL {X  -160.000, Y  +398.523, Z    +0.000, E1   -22.265, E3 +98055.074}
SPL {X  -160.000, Y  +411.325, Z    +0.000, E1   -44.857, E3 +98056.740}
SPL {X  -160.000, Y  +459.786, Z    +0.000, E1   -66.828, E3 +98072.133}
SPL {X  -160.000, Y  +650.407, Z    +0.000, E1   -71.387, E3 +98174.790}
SPL {X  -159.770, Y  +682.971, Z    +0.000, E1   -71.362, E3 +98198.365}
SPL {X  -156.288, Y  +708.665, Z    +0.000, E1   -70.996, E3 +98220.375}
SPL {X  -150.837, Y  +727.770, Z    +0.000, E1   -70.337, E3 +98239.709}
SPL {X  -144.661, Y  +742.760, Z    +0.000, E1   -69.570, E3 +98256.467}
SPL {X  -137.606, Y  +756.037, Z    +0.000, E1   -68.631, E3 +98272.432}
SPL {X  -131.907, Y  +764.957, Z    +0.000, E1   -67.736, E3 +98283.727}
SPL {X  -127.608, Y  +770.921, Z    +0.000, E1   -67.067, E3 +98291.345}
SPL {X  -124.072, Y  +775.426, Z    +0.000, E1   -66.459, E3 +98297.126}
SPL {X   -86.375, Y  +809.082, Z    +0.000, E1   -54.606, E3 +98421.456}
ENDSPLINE

SPLINE
SPL {X  -131.819, Y  +765.085, Z    +0.000, E1   -48.689, E3 +98577.349}
SPL {X  -153.047, Y  +721.053, Z    +0.000, E1   -34.410, E3 +98597.215}
SPL {X  -159.196, Y  +690.423, Z    +0.000, E1   -15.522, E3 +98602.312}
SPL {X  -160.000, Y  +672.957, Z    +0.000, E1    -0.766, E3 +98603.214}
SPL {X  -160.000, Y  +670.573, Z    +0.000, E1    +3.229, E3 +98603.242}
SPL {X  -160.000, Y  +665.683, Z    +0.000, E1   +13.339, E3 +98603.411}
SPL {X  -160.000, Y  +658.186, Z    +0.000, E1   +29.314, E3 +98604.015}
SPL {X  -160.000, Y  +642.169, Z    +0.000, E1   +52.097, E3 +98606.541}
SPL {X  -160.000, Y  +581.106, Z    +0.000, E1   +69.111, E3 +98627.413}
SPL {X  -160.000, Y  +418.281, Z    +0.000, E1   +71.209, E3 +98718.763}
SPL {X  -153.877, Y  +341.861, Z    +0.000, E1   +74.632, E3 +98732.176}
SPL {X  -152.649, Y  +337.758, Z    +0.000, E1   +72.728, E3 +98753.839}
SPL {X  -150.568, Y  +331.578, Z    +0.000, E1   +70.963, E3 +98773.765}
SPL {X  -147.367, Y  +323.387, Z    +0.000, E1   +69.846, E3 +98788.385}
SPL {X  -143.458, Y  +314.849, Z    +0.000, E1   +69.330, E3 +98798.267}
SPL {X  -137.919, Y  +304.592, Z    +0.000, E1   +68.645, E3 +98810.556}
SPL {X  -132.252, Y  +295.648, Z    +0.000, E1   +67.759, E3 +98821.871}
SPL {X  -127.852, Y  +289.504, Z    +0.000, E1   +67.080, E3 +98829.703}
SPL {X  -124.264, Y  +284.911, Z    +0.000, E1   +66.468, E3 +98835.599}
SPL {X   -87.531, Y  +251.766, Z    +0.000, E1   +54.242, E3 +98963.916}
ENDSPLINE

SPLINE
SPL {X  -130.414, Y  +293.006, Z    +0.000, E1   +48.816, E3 +99112.528}
SPL {X  -151.093, Y  +333.061, Z    +0.000, E1   +36.955, E3 +99133.809}
SPL {X  -158.896, Y  +366.939, Z    +0.000, E1   +17.535, E3 +99140.348}
SPL {X  -160.000, Y  +387.267, Z    +0.000, E1    +0.577, E3 +99141.538}
SPL {X  -160.000, Y  +391.471, Z    +0.000, E1    -7.208, E3 +99141.619}
SPL {X  -160.000, Y  +398.523, Z    +0.000, E1   -22.265, E3 +99142.031}
SPL {X  -160.000, Y  +411.325, Z    +0.000, E1   -44.857, E3 +99143.697}
SPL {X  -160.000, Y  +459.786, Z    +0.000, E1   -66.828, E3 +99159.090}
SPL {X  -160.000, Y  +650.407, Z    +0.000, E1   -71.387, E3 +99261.747}
SPL {X  -159.770, Y  +682.971, Z    +0.000, E1   -71.362, E3 +99285.322}
SPL {X  -156.288, Y  +708.665, Z    +0.000, E1   -70.996, E3 +99307.332}
SPL {X  -150.837, Y  +727.770, Z    +0.000, E1   -70.337, E3 +99326.666}
SPL {X  -144.661, Y  +742.760, Z    +0.000, E1   -69.570, E3 +99343.424}
SPL {X  -137.606, Y  +756.037, Z    +0.000, E1   -68.631, E3 +99359.389}
SPL {X  -131.907, Y  +764.957, Z    +0.000, E1   -67.736, E3 +99370.684}
SPL {X  -127.608, Y  +770.921, Z    +0.000, E1   -67.067, E3 +99378.303}
SPL {X  -124.072, Y  +775.426, Z    +0.000, E1   -66.459, E3 +99384.083}
SPL {X   -86.375, Y  +809.082, Z    +0.000, E1   -54.606, E3 +99508.413}
ENDSPLINE

SPLINE
SPL {X  -131.819, Y  +765.085, Z    +0.000, E1   -48.689, E3 +99664.307}
SPL {X  -153.047, Y  +721.053, Z    +0.000, E1   -34.410, E3 +99684.173}
SPL {X  -159.196, Y  +690.423, Z    +0.000, E1   -15.522, E3 +99689.269}
SPL {X  -160.000, Y  +672.957, Z    +0.000, E1    -0.766, E3 +99690.171}
SPL {X  -160.000, Y  +670.573, Z    +0.000, E1    +3.229, E3 +99690.199}
SPL {X  -160.000, Y  +665.683, Z    +0.000, E1   +13.339, E3 +99690.368}
SPL {X  -160.000, Y  +658.186, Z    +0.000, E1   +29.314, E3 +99690.972}
SPL {X  -160.000, Y  +642.169, Z    +0.000, E1   +52.097, E3 +99693.498}
SPL {X  -160.000, Y  +581.106, Z    +0.000, E1   +69.111, E3 +99714.370}
SPL {X  -160.000, Y  +418.281, Z    +0.000, E1   +71.209, E3 +99805.720}
SPL {X  -153.877, Y  +341.861, Z    +0.000, E1   +74.632, E3 +99819.133}
SPL {X  -152.649, Y  +337.758, Z    +0.000, E1   +72.728, E3 +99840.796}
SPL {X  -150.568, Y  +331.578, Z    +0.000, E1   +70.963, E3 +99860.722}
SPL {X  -147.367, Y  +323.387, Z    +0.000, E1   +69.846, E3 +99875.342}
SPL {X  -143.458, Y  +314.849, Z    +0.000, E1   +69.330, E3 +99885.224}
SPL {X  -137.919, Y  +304.592, Z    +0.000, E1   +68.645, E3 +99897.513}
SPL {X  -132.252, Y  +295.648, Z    +0.000, E1   +67.759, E3 +99908.828}
SPL {X  -127.852, Y  +289.504, Z    +0.000, E1   +67.080, E3 +99916.660}
SPL {X  -124.264, Y  +284.911, Z    +0.000, E1   +66.468, E3 +99922.556}
SPL {X   -87.531, Y  +251.766, Z    +0.000, E1   +54.242, E3 +100050.873}
ENDSPLINE

SPLINE
SPL {X  -130.414, Y  +293.006, Z    +0.000, E1   +48.816, E3 +100199.485}
SPL {X  -151.093, Y  +333.061, Z    +0.000, E1   +36.955, E3 +100220.766}
SPL {X  -158.896, Y  +366.939, Z    +0.000, E1   +17.535, E3 +100227.305}
SPL {X  -160.000, Y  +387.267, Z    +0.000, E1    +0.577, E3 +100228.495}
SPL {X  -160.000, Y  +391.471, Z    +0.000, E1    -7.208, E3 +100228.576}
SPL {X  -160.000, Y  +398.523, Z    +0.000, E1   -22.265, E3 +100228.988}
SPL {X  -160.000, Y  +411.325, Z    +0.000, E1   -44.857, E3 +100230.654}
SPL {X  -160.000, Y  +459.786, Z    +0.000, E1   -66.828, E3 +100246.047}
SPL {X  -160.000, Y  +650.407, Z    +0.000, E1   -71.387, E3 +100348.704}
SPL {X  -159.770, Y  +682.971, Z    +0.000, E1   -71.362, E3 +100372.279}
SPL {X  -156.288, Y  +708.665, Z    +0.000, E1   -70.996, E3 +100394.289}
SPL {X  -150.837, Y  +727.770, Z    +0.000, E1   -70.337, E3 +100413.623}
SPL {X  -144.661, Y  +742.760, Z    +0.000, E1   -69.570, E3 +100430.381}
SPL {X  -137.606, Y  +756.037, Z    +0.000, E1   -68.631, E3 +100446.346}
SPL {X  -131.907, Y  +764.957, Z    +0.000, E1   -67.736, E3 +100457.641}
SPL {X  -127.608, Y  +770.921, Z    +0.000, E1   -67.067, E3 +100465.260}
SPL {X  -124.072, Y  +775.426, Z    +0.000, E1   -66.459, E3 +100471.040}
SPL {X   -86.375, Y  +809.082, Z    +0.000, E1   -54.606, E3 +100595.370}
ENDSPLINE

SPLINE
SPL {X  -131.819, Y  +765.085, Z    +0.000, E1   -48.689, E3 +100751.264}
SPL {X  -153.047, Y  +721.053, Z    +0.000, E1   -34.410, E3 +100771.130}
SPL {X  -159.196, Y  +690.423, Z    +0.000, E1   -15.522, E3 +100776.226}
SPL {X  -160.000, Y  +672.957, Z    +0.000, E1    -0.766, E3 +100777.128}
SPL {X  -160.000, Y  +670.573, Z    +0.000, E1    +3.229, E3 +100777.156}
SPL {X  -160.000, Y  +665.683, Z    +0.000, E1   +13.339, E3 +100777.325}
SPL {X  -160.000, Y  +658.186, Z    +0.000, E1   +29.314, E3 +100777.930}
SPL {X  -160.000, Y  +642.169, Z    +0.000, E1   +52.097, E3 +100780.455}
SPL {X  -160.000, Y  +581.106, Z    +0.000, E1   +69.111, E3 +100801.327}
SPL {X  -160.000, Y  +418.281, Z    +0.000, E1   +71.209, E3 +100892.677}
SPL {X  -153.877, Y  +341.861, Z    +0.000, E1   +74.632, E3 +100906.090}
SPL {X  -152.649, Y  +337.758, Z    +0.000, E1   +72.728, E3 +100927.753}
SPL {X  -150.568, Y  +331.578, Z    +0.000, E1   +70.963, E3 +100947.679}
SPL {X  -147.367, Y  +323.387, Z    +0.000, E1   +69.846, E3 +100962.299}
SPL {X  -143.458, Y  +314.849, Z    +0.000, E1   +69.330, E3 +100972.182}
SPL {X  -137.919, Y  +304.592, Z    +0.000, E1   +68.645, E3 +100984.470}
SPL {X  -132.252, Y  +295.648, Z    +0.000, E1   +67.759, E3 +100995.785}
SPL {X  -127.852, Y  +289.504, Z    +0.000, E1   +67.080, E3 +101003.617}
SPL {X  -124.264, Y  +284.911, Z    +0.000, E1   +66.468, E3 +101009.513}
SPL {X   -87.531, Y  +251.766, Z    +0.000, E1   +54.242, E3 +101137.830}
ENDSPLINE

SPLINE
SPL {X  -130.414, Y  +293.006, Z    +0.000, E1   +48.816, E3 +101286.442}
SPL {X  -151.093, Y  +333.061, Z    +0.000, E1   +36.955, E3 +101307.723}
SPL {X  -158.896, Y  +366.939, Z    +0.000, E1   +17.535, E3 +101314.263}
SPL {X  -160.000, Y  +387.267, Z    +0.000, E1    +0.577, E3 +101315.452}
SPL {X  -160.000, Y  +391.471, Z    +0.000, E1    -7.208, E3 +101315.533}
SPL {X  -160.000, Y  +398.523, Z    +0.000, E1   -22.265, E3 +101315.945}
SPL {X  -160.000, Y  +411.325, Z    +0.000, E1   -44.857, E3 +101317.611}
SPL {X  -160.000, Y  +459.786, Z    +0.000, E1   -66.828, E3 +101333.004}
SPL {X  -160.000, Y  +650.407, Z    +0.000, E1   -71.387, E3 +101435.661}
SPL {X  -159.770, Y  +682.971, Z    +0.000, E1   -71.362, E3 +101459.236}
SPL {X  -156.288, Y  +708.665, Z    +0.000, E1   -70.996, E3 +101481.247}
SPL {X  -150.837, Y  +727.770, Z    +0.000, E1   -70.337, E3 +101500.580}
SPL {X  -144.661, Y  +742.760, Z    +0.000, E1   -69.570, E3 +101517.338}
SPL {X  -137.606, Y  +756.037, Z    +0.000, E1   -68.631, E3 +101533.303}
SPL {X  -131.907, Y  +764.957, Z    +0.000, E1   -67.736, E3 +101544.598}
SPL {X  -127.608, Y  +770.921, Z    +0.000, E1   -67.067, E3 +101552.217}
SPL {X  -124.072, Y  +775.426, Z    +0.000, E1   -66.459, E3 +101557.997}
SPL {X   -86.375, Y  +809.082, Z    +0.000, E1   -54.606, E3 +101682.327}
ENDSPLINE

SPLINE
SPL {X  -131.819, Y  +765.085, Z    +0.000, E1   -48.689, E3 +101838.221}
SPL {X  -153.047, Y  +721.053, Z    +0.000, E1   -34.410, E3 +101858.087}
SPL {X  -159.196, Y  +690.423, Z    +0.000, E1   -15.522, E3 +101863.183}
SPL {X  -160.000, Y  +672.957, Z    +0.000, E1    -0.766, E3 +101864.085}
SPL {X  -160.000, Y  +670.573, Z    +0.000, E1    +3.229, E3 +101864.113}
SPL {X  -160.000, Y  +665.683, Z    +0.000, E1   +13.339, E3 +101864.282}
SPL {X  -160.000, Y  +658.186, Z    +0.000, E1   +29.314, E3 +101864.887}
SPL {X  -160.000, Y  +642.169, Z    +0.000, E1   +52.097, E3 +101867.412}
SPL {X  -160.000, Y  +581.106, Z    +0.000, E1   +69.111, E3 +101888.284}
SPL {X  -160.000, Y  +418.281, Z    +0.000, E1   +71.209, E3 +101979.634}
SPL {X  -153.877, Y  +341.861, Z    +0.000, E1   +74.632, E3 +101993.048}
SPL {X  -152.649, Y  +337.758, Z    +0.000, E1   +72.728, E3 +102014.710}
SPL {X  -150.568, Y  +331.578, Z    +0.000, E1   +70.963, E3 +102034.636}
SPL {X  -147.367, Y  +323.387, Z    +0.000, E1   +69.846, E3 +102049.256}
SPL {X  -143.458, Y  +314.849, Z    +0.000, E1   +69.330, E3 +102059.139}
SPL {X  -137.919, Y  +304.592, Z    +0.000, E1   +68.645, E3 +102071.427}
SPL {X  -132.252, Y  +295.648, Z    +0.000, E1   +67.759, E3 +102082.742}
SPL {X  -127.852, Y  +289.504, Z    +0.000, E1   +67.080, E3 +102090.574}
SPL {X  -124.264, Y  +284.911, Z    +0.000, E1   +66.468, E3 +102096.470}
SPL {X   -87.531, Y  +251.766, Z    +0.000, E1   +54.242, E3 +102224.787}
ENDSPLINE

SPLINE
SPL {X  -130.414, Y  +293.006, Z    +0.000, E1   +48.816, E3 +102373.399}
SPL {X  -151.093, Y  +333.061, Z    +0.000, E1   +36.955, E3 +102394.680}
SPL {X  -158.896, Y  +366.939, Z    +0.000, E1   +17.535, E3 +102401.220}
SPL {X  -160.000, Y  +387.267, Z    +0.000, E1    +0.577, E3 +102402.409}
SPL {X  -160.000, Y  +391.471, Z    +0.000, E1    -7.208, E3 +102402.490}
SPL {X  -160.000, Y  +398.523, Z    +0.000, E1   -22.265, E3 +102402.902}
SPL {X  -160.000, Y  +411.325, Z    +0.000, E1   -44.857, E3 +102404.568}
SPL {X  -160.000, Y  +459.786, Z    +0.000, E1   -66.828, E3 +102419.961}
SPL {X  -160.000, Y  +650.407, Z    +0.000, E1   -71.387, E3 +102522.618}
SPL {X  -159.770, Y  +682.971, Z    +0.000, E1   -71.362, E3 +102546.193}
SPL {X  -156.288, Y  +708.665, Z    +0.000, E1   -70.996, E3 +102568.204}
SPL {X  -150.837, Y  +727.770, Z    +0.000, E1   -70.337, E3 +102587.537}
SPL {X  -144.661, Y  +742.760, Z    +0.000, E1   -69.570, E3 +102604.296}
SPL {X  -137.606, Y  +756.037, Z    +0.000, E1   -68.631, E3 +102620.260}
SPL {X  -131.907, Y  +764.957, Z    +0.000, E1   -67.736, E3 +102631.555}
SPL {X  -127.608, Y  +770.921, Z    +0.000, E1   -67.067, E3 +102639.174}
SPL {X  -124.072, Y  +775.426, Z    +0.000, E1   -66.459, E3 +102644.954}
SPL {X   -86.375, Y  +809.082, Z    +0.000, E1   -54.606, E3 +102769.284}
ENDSPLINE

SPLINE
SPL {X  -131.819, Y  +765.085, Z    +0.000, E1   -48.689, E3 +102925.178}
SPL {X  -153.047, Y  +721.053, Z    +0.000, E1   -34.410, E3 +102945.044}
SPL {X  -159.196, Y  +690.423, Z    +0.000, E1   -15.522, E3 +102950.140}
SPL {X  -160.000, Y  +672.957, Z    +0.000, E1    -0.766, E3 +102951.042}
SPL {X  -160.000, Y  +670.573, Z    +0.000, E1    +3.229, E3 +102951.070}
SPL {X  -160.000, Y  +665.683, Z    +0.000, E1   +13.339, E3 +102951.240}
SPL {X  -160.000, Y  +658.186, Z    +0.000, E1   +29.314, E3 +102951.844}
SPL {X  -160.000, Y  +642.169, Z    +0.000, E1   +52.097, E3 +102954.369}
SPL {X  -160.000, Y  +581.106, Z    +0.000, E1   +69.111, E3 +102975.242}
SPL {X  -160.000, Y  +418.281, Z    +0.000, E1   +71.209, E3 +103066.591}
SPL {X  -153.877, Y  +341.861, Z    +0.000, E1   +74.632, E3 +103080.005}
SPL {X  -152.649, Y  +337.758, Z    +0.000, E1   +72.728, E3 +103101.667}
SPL {X  -150.568, Y  +331.578, Z    +0.000, E1   +70.963, E3 +103121.593}
SPL {X  -147.367, Y  +323.387, Z    +0.000, E1   +69.846, E3 +103136.214}
SPL {X  -143.458, Y  +314.849, Z    +0.000, E1   +69.330, E3 +103146.096}
SPL {X  -137.919, Y  +304.592, Z    +0.000, E1   +68.645, E3 +103158.385}
SPL {X  -132.252, Y  +295.648, Z    +0.000, E1   +67.759, E3 +103169.699}
SPL {X  -127.852, Y  +289.504, Z    +0.000, E1   +67.080, E3 +103177.532}
SPL {X  -124.264, Y  +284.911, Z    +0.000, E1   +66.468, E3 +103183.427}
SPL {X   -87.531, Y  +251.766, Z    +0.000, E1   +54.242, E3 +103311.744}
ENDSPLINE

SPLINE
SPL {X  -130.414, Y  +293.006, Z    +0.000, E1   +48.816, E3 +103460.356}
SPL {X  -151.093, Y  +333.061, Z    +0.000, E1   +36.955, E3 +103481.637}
SPL {X  -158.896, Y  +366.939, Z    +0.000, E1   +17.535, E3 +103488.177}
SPL {X  -160.000, Y  +387.267, Z    +0.000, E1    +0.577, E3 +103489.367}
SPL {X  -160.000, Y  +391.471, Z    +0.000, E1    -7.208, E3 +103489.448}
SPL {X  -160.000, Y  +398.523, Z    +0.000, E1   -22.265, E3 +103489.859}
SPL {X  -160.000, Y  +411.325, Z    +0.000, E1   -44.857, E3 +103491.525}
SPL {X  -160.000, Y  +459.786, Z    +0.000, E1   -66.828, E3 +103506.918}
SPL {X  -160.000, Y  +650.407, Z    +0.000, E1   -71.387, E3 +103609.575}
SPL {X  -159.770, Y  +682.971, Z    +0.000, E1   -71.362, E3 +103633.151}
SPL {X  -156.288, Y  +708.665, Z    +0.000, E1   -70.996, E3 +103655.161}
SPL {X  -150.837, Y  +727.770, Z    +0.000, E1   -70.337, E3 +103674.494}
SPL {X  -144.661, Y  +742.760, Z    +0.000, E1   -69.570, E3 +103691.253}
SPL {X  -137.606, Y  +756.037, Z    +0.000, E1   -68.631, E3 +103707.217}
SPL {X  -131.907, Y  +764.957, Z    +0.000, E1   -67.736, E3 +103718.512}
SPL {X  -127.608, Y  +770.921, Z    +0.000, E1   -67.067, E3 +103726.131}
SPL {X  -124.072, Y  +775.426, Z    +0.000, E1   -66.459, E3 +103731.911}
SPL {X   -86.375, Y  +809.082, Z    +0.000, E1   -54.606, E3 +103856.242}
ENDSPLINE

SPLINE
SPL {X  -131.819, Y  +765.085, Z    +0.000, E1   -48.689, E3 +104012.135}
SPL {X  -153.047, Y  +721.053, Z    +0.000, E1   -34.410, E3 +104032.001}
SPL {X  -159.196, Y  +690.423, Z    +0.000, E1   -15.522, E3 +104037.097}
SPL {X  -160.000, Y  +672.957, Z    +0.000, E1    -0.766, E3 +104037.999}
SPL {X  -160.000, Y  +670.573, Z    +0.000, E1    +3.229, E3 +104038.027}
SPL {X  -160.000, Y  +665.683, Z    +0.000, E1   +13.339, E3 +104038.197}
SPL {X  -160.000, Y  +658.186, Z    +0.000, E1   +29.314, E3 +104038.801}
SPL {X  -160.000, Y  +642.169, Z    +0.000, E1   +52.097, E3 +104041.326}
SPL {X  -160.000, Y  +581.106, Z    +0.000, E1   +69.111, E3 +104062.199}
SPL {X  -160.000, Y  +418.281, Z    +0.000, E1   +71.209, E3 +104153.548}
SPL {X  -153.877, Y  +341.861, Z    +0.000, E1   +74.632, E3 +104166.962}
SPL {X  -152.649, Y  +337.758, Z    +0.000, E1   +72.728, E3 +104188.624}
SPL {X  -150.568, Y  +331.578, Z    +0.000, E1   +70.963, E3 +104208.550}
SPL {X  -147.367, Y  +323.387, Z    +0.000, E1   +69.846, E3 +104223.171}
SPL {X  -143.458, Y  +314.849, Z    +0.000, E1   +69.330, E3 +104233.053}
SPL {X  -137.919, Y  +304.592, Z    +0.000, E1   +68.645, E3 +104245.342}
SPL {X  -132.252, Y  +295.648, Z    +0.000, E1   +67.759, E3 +104256.656}
SPL {X  -127.852, Y  +289.504, Z    +0.000, E1   +67.080, E3 +104264.489}
SPL {X  -124.264, Y  +284.911, Z    +0.000, E1   +66.468, E3 +104270.385}
SPL {X   -87.531, Y  +251.766, Z    +0.000, E1   +54.242, E3 +104398.701}
ENDSPLINE

SPLINE
SPL {X  -130.414, Y  +293.006, Z    +0.000, E1   +48.816, E3 +104547.314}
SPL {X  -151.093, Y  +333.061, Z    +0.000, E1   +36.955, E3 +104568.594}
SPL {X  -158.896, Y  +366.939, Z    +0.000, E1   +17.535, E3 +104575.134}
SPL {X  -160.000, Y  +387.267, Z    +0.000, E1    +0.577, E3 +104576.324}
SPL {X  -160.000, Y  +391.471, Z    +0.000, E1    -7.208, E3 +104576.405}
SPL {X  -160.000, Y  +398.523, Z    +0.000, E1   -22.265, E3 +104576.817}
SPL {X  -160.000, Y  +411.325, Z    +0.000, E1   -44.857, E3 +104578.482}
SPL {X  -160.000, Y  +459.786, Z    +0.000, E1   -66.828, E3 +104593.875}
SPL {X  -160.000, Y  +650.407, Z    +0.000, E1   -71.387, E3 +104696.532}
SPL {X  -159.770, Y  +682.971, Z    +0.000, E1   -71.362, E3 +104720.108}
SPL {X  -156.288, Y  +708.665, Z    +0.000, E1   -70.996, E3 +104742.118}
SPL {X  -150.837, Y  +727.770, Z    +0.000, E1   -70.337, E3 +104761.452}
SPL {X  -144.661, Y  +742.760, Z    +0.000, E1   -69.570, E3 +104778.210}
SPL {X  -137.606, Y  +756.037, Z    +0.000, E1   -68.631, E3 +104794.175}
SPL {X  -131.907, Y  +764.957, Z    +0.000, E1   -67.736, E3 +104805.470}
SPL {X  -127.608, Y  +770.921, Z    +0.000, E1   -67.067, E3 +104813.088}
SPL {X  -124.072, Y  +775.426, Z    +0.000, E1   -66.459, E3 +104818.868}
SPL {X   -86.375, Y  +809.082, Z    +0.000, E1   -54.606, E3 +104943.199}
ENDSPLINE

SPLINE
SPL {X  -131.819, Y  +765.085, Z    +0.000, E1   -48.689, E3 +105099.092}
SPL {X  -153.047, Y  +721.053, Z    +0.000, E1   -34.410, E3 +105118.958}
SPL {X  -159.196, Y  +690.423, Z    +0.000, E1   -15.522, E3 +105124.055}
SPL {X  -160.000, Y  +672.957, Z    +0.000, E1    -0.766, E3 +105124.956}
SPL {X  -160.000, Y  +670.573, Z    +0.000, E1    +3.229, E3 +105124.985}
SPL {X  -160.000, Y  +665.683, Z    +0.000, E1   +13.339, E3 +105125.154}
SPL {X  -160.000, Y  +658.186, Z    +0.000, E1   +29.314, E3 +105125.758}
SPL {X  -160.000, Y  +642.169, Z    +0.000, E1   +52.097, E3 +105128.284}
SPL {X  -160.000, Y  +581.106, Z    +0.000, E1   +69.111, E3 +105149.156}
SPL {X  -160.000, Y  +418.281, Z    +0.000, E1   +71.209, E3 +105240.505}
SPL {X  -153.877, Y  +341.861, Z    +0.000, E1   +74.632, E3 +105253.919}
SPL {X  -152.649, Y  +337.758, Z    +0.000, E1   +72.728, E3 +105275.582}
SPL {X  -150.568, Y  +331.578, Z    +0.000, E1   +70.963, E3 +105295.507}
SPL {X  -147.367, Y  +323.387, Z    +0.000, E1   +69.846, E3 +105310.128}
SPL {X  -143.458, Y  +314.849, Z    +0.000, E1   +69.330, E3 +105320.010}
SPL {X  -137.919, Y  +304.592, Z    +0.000, E1   +68.645, E3 +105332.299}
SPL {X  -132.252, Y  +295.648, Z    +0.000, E1   +67.759, E3 +105343.614}
SPL {X  -127.852, Y  +289.504, Z    +0.000, E1   +67.080, E3 +105351.446}
SPL {X  -124.264, Y  +284.911, Z    +0.000, E1   +66.468, E3 +105357.342}
SPL {X   -87.531, Y  +251.766, Z    +0.000, E1   +54.242, E3 +105485.658}
ENDSPLINE

SPLINE
SPL {X  -130.414, Y  +293.006, Z    +0.000, E1   +48.816, E3 +105634.271}
SPL {X  -151.093, Y  +333.061, Z    +0.000, E1   +36.955, E3 +105655.551}
SPL {X  -158.896, Y  +366.939, Z    +0.000, E1   +17.535, E3 +105662.091}
SPL {X  -160.000, Y  +387.267, Z    +0.000, E1    +0.577, E3 +105663.281}
SPL {X  -160.000, Y  +391.471, Z    +0.000, E1    -7.208, E3 +105663.362}
SPL {X  -160.000, Y  +398.523, Z    +0.000, E1   -22.265, E3 +105663.774}
SPL {X  -160.000, Y  +411.325, Z    +0.000, E1   -44.857, E3 +105665.439}
SPL {X  -160.000, Y  +459.786, Z    +0.000, E1   -66.828, E3 +105680.832}
SPL {X  -160.000, Y  +650.407, Z    +0.000, E1   -71.387, E3 +105783.489}
SPL {X  -159.770, Y  +682.971, Z    +0.000, E1   -71.362, E3 +105807.065}
SPL {X  -156.288, Y  +708.665, Z    +0.000, E1   -70.996, E3 +105829.075}
SPL {X  -150.837, Y  +727.770, Z    +0.000, E1   -70.337, E3 +105848.409}
SPL {X  -144.661, Y  +742.760, Z    +0.000, E1   -69.570, E3 +105865.167}
SPL {X  -137.606, Y  +756.037, Z    +0.000, E1   -68.631, E3 +105881.132}
SPL {X  -131.907, Y  +764.957, Z    +0.000, E1   -67.736, E3 +105892.427}
SPL {X  -127.608, Y  +770.921, Z    +0.000, E1   -67.067, E3 +105900.045}
SPL {X  -124.072, Y  +775.426, Z    +0.000, E1   -66.459, E3 +105905.826}
SPL {X   -86.375, Y  +809.082, Z    +0.000, E1   -54.606, E3 +106030.156}
ENDSPLINE

SPLINE
SPL {X  -131.819, Y  +765.085, Z    +0.000, E1   -48.689, E3 +106186.049}
SPL {X  -153.047, Y  +721.053, Z    +0.000, E1   -34.410, E3 +106205.915}
SPL {X  -159.196, Y  +690.423, Z    +0.000, E1   -15.522, E3 +106211.012}
SPL {X  -160.000, Y  +672.957, Z    +0.000, E1    -0.766, E3 +106211.914}
SPL {X  -160.000, Y  +670.573, Z    +0.000, E1    +3.229, E3 +106211.942}
SPL {X  -160.000, Y  +665.683, Z    +0.000, E1   +13.339, E3 +106212.111}
SPL {X  -160.000, Y  +658.186, Z    +0.000, E1   +29.314, E3 +106212.715}
SPL {X  -160.000, Y  +642.169, Z    +0.000, E1   +52.097, E3 +106215.241}
SPL {X  -160.000, Y  +581.106, Z    +0.000, E1   +69.111, E3 +106236.113}
SPL {X  -160.000, Y  +418.281, Z    +0.000, E1   +71.209, E3 +106327.462}
SPL {X  -153.877, Y  +341.861, Z    +0.000, E1   +74.632, E3 +106340.876}
SPL {X  -152.649, Y  +337.758, Z    +0.000, E1   +72.728, E3 +106362.539}
SPL {X  -150.568, Y  +331.578, Z    +0.000, E1   +70.963, E3 +106382.465}
SPL {X  -147.367, Y  +323.387, Z    +0.000, E1   +69.846, E3 +106397.085}
SPL {X  -143.458, Y  +314.849, Z    +0.000, E1   +69.330, E3 +106406.967}
SPL {X  -137.919, Y  +304.592, Z    +0.000, E1   +68.645, E3 +106419.256}
SPL {X  -132.252, Y  +295.648, Z    +0.000, E1   +67.759, E3 +106430.571}
SPL {X  -127.852, Y  +289.504, Z    +0.000, E1   +67.080, E3 +106438.403}
SPL {X  -124.264, Y  +284.911, Z    +0.000, E1   +66.468, E3 +106444.299}
SPL {X   -87.531, Y  +251.766, Z    +0.000, E1   +54.242, E3 +106572.615}
ENDSPLINE

SPLINE
SPL {X  -130.414, Y  +293.006, Z    +0.000, E1   +48.816, E3 +106721.228}
SPL {X  -151.093, Y  +333.061, Z    +0.000, E1   +36.955, E3 +106742.508}
SPL {X  -158.896, Y  +366.939, Z    +0.000, E1   +17.535, E3 +106749.048}
SPL {X  -160.000, Y  +387.267, Z    +0.000, E1    +0.577, E3 +106750.238}
SPL {X  -160.000, Y  +391.471, Z    +0.000, E1    -7.208, E3 +106750.319}
SPL {X  -160.000, Y  +398.523, Z    +0.000, E1   -22.265, E3 +106750.731}
SPL {X  -160.000, Y  +411.325, Z    +0.000, E1   -44.857, E3 +106752.397}
SPL {X  -160.000, Y  +459.786, Z    +0.000, E1   -66.828, E3 +106767.789}
SPL {X  -160.000, Y  +650.407, Z    +0.000, E1   -71.387, E3 +106870.446}
SPL {X  -159.770, Y  +682.971, Z    +0.000, E1   -71.362, E3 +106894.022}
SPL {X  -156.288, Y  +708.665, Z    +0.000, E1   -70.996, E3 +106916.032}
SPL {X  -150.837, Y  +727.770, Z    +0.000, E1   -70.337, E3 +106935.366}
SPL {X  -144.661, Y  +742.760, Z    +0.000, E1   -69.570, E3 +106952.124}
SPL {X  -137.606, Y  +756.037, Z    +0.000, E1   -68.631, E3 +106968.089}
SPL {X  -131.907, Y  +764.957, Z    +0.000, E1   -67.736, E3 +106979.384}
SPL {X  -127.608, Y  +770.921, Z    +0.000, E1   -67.067, E3 +106987.002}
SPL {X  -124.072, Y  +775.426, Z    +0.000, E1   -66.459, E3 +106992.783}
SPL {X   -86.375, Y  +809.082, Z    +0.000, E1   -54.606, E3 +107117.113}
ENDSPLINE

SPLINE
SPL {X  -131.819, Y  +765.085, Z    +0.000, E1   -48.689, E3 +107273.006}
SPL {X  -153.047, Y  +721.053, Z    +0.000, E1   -34.410, E3 +107292.872}
SPL {X  -159.196, Y  +690.423, Z    +0.000, E1   -15.522, E3 +107297.969}
SPL {X  -160.000, Y  +672.957, Z    +0.000, E1    -0.766, E3 +107298.871}
SPL {X  -160.000, Y  +670.573, Z    +0.000, E1    +3.229, E3 +107298.899}
SPL {X  -160.000, Y  +665.683, Z    +0.000, E1   +13.339, E3 +107299.068}
SPL {X  -160.000, Y  +658.186, Z    +0.000, E1   +29.314, E3 +107299.672}
SPL {X  -160.000, Y  +642.169, Z    +0.000, E1   +52.097, E3 +107302.198}
SPL {X  -160.000, Y  +581.106, Z    +0.000, E1   +69.111, E3 +107323.070}
SPL {X  -160.000, Y  +418.281, Z    +0.000, E1   +71.209, E3 +107414.420}
SPL {X  -153.877, Y  +341.861, Z    +0.000, E1   +74.632, E3 +107427.833}
SPL {X  -152.649, Y  +337.758, Z    +0.000, E1   +72.728, E3 +107449.496}
SPL {X  -150.568, Y  +331.578, Z    +0.000, E1   +70.963, E3 +107469.422}
SPL {X  -147.367, Y  +323.387, Z    +0.000, E1   +69.846, E3 +107484.042}
SPL {X  -143.458, Y  +314.849, Z    +0.000, E1   +69.330, E3 +107493.924}
SPL {X  -137.919, Y  +304.592, Z    +0.000, E1   +68.645, E3 +107506.213}
SPL {X  -132.252, Y  +295.648, Z    +0.000, E1   +67.759, E3 +107517.528}
SPL {X  -127.852, Y  +289.504, Z    +0.000, E1   +67.080, E3 +107525.360}
SPL {X  -124.264, Y  +284.911, Z    +0.000, E1   +66.468, E3 +107531.256}
SPL {X   -87.531, Y  +251.766, Z    +0.000, E1   +54.242, E3 +107659.573}
ENDSPLINE

SPLINE
SPL {X  -130.414, Y  +293.006, Z    +0.000, E1   +48.816, E3 +107808.185}
SPL {X  -151.093, Y  +333.061, Z    +0.000, E1   +36.955, E3 +107829.466}
SPL {X  -158.896, Y  +366.939, Z    +0.000, E1   +17.535, E3 +107836.005}
SPL {X  -160.000, Y  +387.267, Z    +0.000, E1    +0.577, E3 +107837.195}
SPL {X  -160.000, Y  +391.471, Z    +0.000, E1    -7.208, E3 +107837.276}
SPL {X  -160.000, Y  +398.523, Z    +0.000, E1   -22.265, E3 +107837.688}
SPL {X  -160.000, Y  +411.325, Z    +0.000, E1   -44.857, E3 +107839.354}
SPL {X  -160.000, Y  +459.786, Z    +0.000, E1   -66.828, E3 +107854.747}
SPL {X  -160.000, Y  +650.407, Z    +0.000, E1   -71.387, E3 +107957.404}
SPL {X  -159.770, Y  +682.971, Z    +0.000, E1   -71.362, E3 +107980.979}
SPL {X  -156.288, Y  +708.665, Z    +0.000, E1   -70.996, E3 +108002.989}
SPL {X  -150.837, Y  +727.770, Z    +0.000, E1   -70.337, E3 +108022.323}
SPL {X  -144.661, Y  +742.760, Z    +0.000, E1   -69.570, E3 +108039.081}
SPL {X  -137.606, Y  +756.037, Z    +0.000, E1   -68.631, E3 +108055.046}
SPL {X  -131.907, Y  +764.957, Z    +0.000, E1   -67.736, E3 +108066.341}
SPL {X  -127.608, Y  +770.921, Z    +0.000, E1   -67.067, E3 +108073.959}
SPL {X  -124.072, Y  +775.426, Z    +0.000, E1   -66.459, E3 +108079.740}
SPL {X   -86.375, Y  +809.082, Z    +0.000, E1   -54.606, E3 +108204.070}
ENDSPLINE

